KUKA KRL program: EPS_2_251520_SPSOVERFLOW_A_20260212031628.src

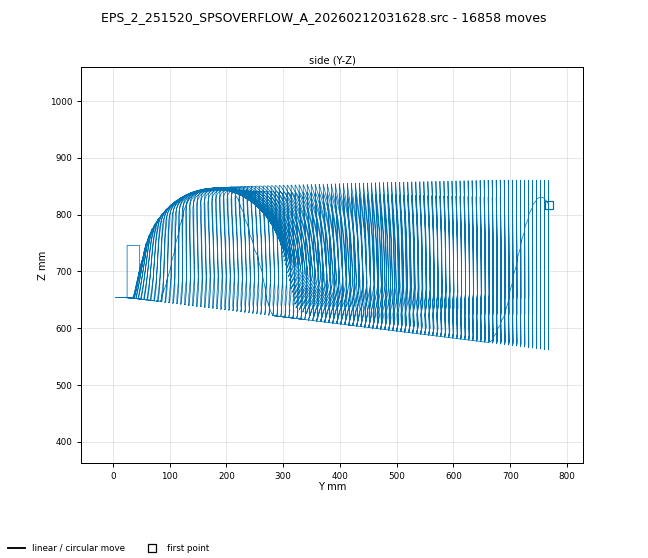
[picture p0: tool path of EPS_2_251520_SPSOVERFLOW_A_20260212031628.src, 16858 of 16860 moves have a stored position in this frame; points joined in program order, loops and branches not executed]
&ACCESS RVP
&REL 4
&COMMENT QRS 19112012
&PARAM EDITMASK = *
DEF PART()
EXT BAS (BAS_COMMAND :IN,REAL :IN )
INT I
BAS (#INITMOV,0 )

;KUKA QRS Post kuka4.cps  Date:22-06-2017 !

File_ID=3026

QRS_PRE_INIT()

;Init var - Until changes are made in qrs_pre_init
Outlet_Square_prg=0
Inlet_1_Square_prg=0
Inlet_2_Square_prg=0
Inlet_3_Square_prg=0
Inlet_4_Square_prg=0
Inlet_5_Square_prg=0

Outlet_1={X 0.000, Y 668.450, Z 760.500, B 0.000, E1 0.000 }
Inlet_1={X 0.000, Y 670.580, Z 730.500, B 0.000, E1 100.000 }
Outlet_1_type=201
Inlet_1_type=201
;QRS#1=Sidecore dimensions
;QRS#2=200-8" PVC SDR 35
;QRS#3=200-8" PVC SDR 35
;QRS#4=
;QRS#5=
;QRS#6=
;QRS#7=
;QRS#8=
;QRS#9=12-08 PSX
;QRS#10=12-08 PSX
;QRS#11=
;QRS#12=
;QRS#13=
;QRS#14=
;QRS#15=
;QRS#16=1524x152x1219 4'
;QRS#17=EPS Height
;QRS#18=861
;QRS#19=*
;QRS#20= UPDATED VERSION 22-06-2017
;QRS#21=*
Outlet_Square=0100
Inlet_1_Square=0100
Inlet_2_Square=0
Inlet_3_Square=0
Inlet_4_Square=0
Inlet_5_Square=0
Mill_Square=1
Outlet_Square_Prg=204
Inlet_1_Square_prg=204

QRS_INIT()

$ADVANCE=5

; T1
PTP {E1 174.142,E2 174.142}
PTP {X 0,Y 767.495,A -85,B 0,C 180,E1 174.142,E2 174.142,E3 0,E4 0,E5 0,E6 0}
QRS_SPEED_INIT()
LIN {X 0,Y 767.495,Z 817.254,A -85,B 0,C 180,E1 174.142,E2 174.142,E3 0,E4 0,E5 0,E6 0} C_VEL
LIN {X 0,Y 767.491,Z 822.732,A -85,B 0,C 180,E1 173.186,E2 173.186} C_VEL
LIN {X 0,Y 767.495,Z 825.01,A -85,B 0,C 180,E1 172.66,E2 172.66} C_VEL
LIN {X 0,Y 767.487,Z 828.448,A -85,B 0,C 180,E1 171.604,E2 171.604} C_VEL
LIN {X 0,Y 767.494,Z 830.063,A -85,B 0,C 180,E1 170.545,E2 170.545} C_VEL
LIN {X 0,Y 767.499,Z 830.375,A -85,B 0,C 180,E1 170.015,E2 170.015} C_VEL
LIN {X 0,Y 767.487,Z 829.609,A -85,B 0,C 180,E1 168.951,E2 168.951} C_VEL
LIN {X 0,Y 767.493,Z 828.662,A -85,B 0,C 180,E1 168.418,E2 168.418} C_VEL
LIN {X 0,Y 767.489,Z 825.435,A -85,B 0,C 180,E1 167.348,E2 167.348} C_VEL
LIN {X 0,Y 767.493,Z 821.811,A -85,B 0,C 180,E1 166.543,E2 166.543} C_VEL
LIN {X 0,Y 767.492,Z 817.014,A -85,B 0,C 180,E1 165.735,E2 165.735} C_VEL
LIN {X 0,Y 767.496,Z 810.871,A -85,B 0,C 180,E1 164.924,E2 164.924} C_VEL
LIN {X 0,Y 767.492,Z 804.595,A -85,B 0,C 180,E1 164.246,E2 164.246} C_VEL
LIN {X 0,Y 767.496,Z 796.955,A -85,B 0,C 180,E1 163.566,E2 163.566} C_VEL
LIN {X 0,Y 767.5,Z 788.629,A -85,B 0,C 180,E1 162.952,E2 162.952} C_VEL
LIN {X 0,Y 767.499,Z 780.947,A -85,B 0,C 180,E1 162.472,E2 162.472} C_VEL
LIN {X 0,Y 767.499,Z 771.732,A -85,B 0,C 180,E1 161.992,E2 161.992} C_VEL
LIN {X 0,Y 767.49,Z 762.141,A -85,B 0,C 180,E1 161.581,E2 161.581} C_VEL
LIN {X 0,Y 767.479,Z 750.832,A -85,B 0,C 180,E1 161.199,E2 161.199} C_VEL
LIN {X 0,Y 767.462,Z 740.016,A -85,B 0,C 180,E1 160.922,E2 160.922} C_VEL
LIN {X 0,Y 767.482,Z 729.744,A -85,B 0,C 180,E1 160.733,E2 160.733} C_VEL
LIN {X 0,Y 767.493,Z 712.465,A -85,B 0,C 180,E1 160.542,E2 160.542} C_VEL
LIN {X 0,Y 767.476,Z 620.271,A -85,B 0,C 180,E1 159.673,E2 159.673} C_VEL
LIN {X 0,Y 767.464,Z 604.056,A -85,B 0,C 180,E1 157.461,E2 157.461} C_VEL
LIN {X 0,Y 767.465,Z 586.448,A -85,B 0,C 180,E1 155.038,E2 155.038} C_VEL
LIN {X 0,Y 767.495,Z 568.677,A -85,B 0,C 180,E1 152.568,E2 152.568} C_VEL
LIN {X 0,Y 767.455,Z 561.691,A -85,B 0,C 180,E1 151.577,E2 151.577} C_VEL
LIN {X 0,Y 767.446,Z 561.687,A -85,B 0,C 180,E1 149.263,E2 149.263} C_VEL
LIN {X 0,Y 767.456,Z 561.684,A -85,B 0,C 180,E1 147.105,E2 147.105} C_VEL
LIN {X 0,Y 767.473,Z 561.68,A -85,B 0,C 180,E1 144.902,E2 144.902} C_VEL
LIN {X 0,Y 767.486,Z 561.692,A -85,B 0,C 180,E1 142.304,E2 142.304} C_VEL
LIN {X 0,Y 767.49,Z 561.702,A -85,B 0,C 180,E1 140.052,E2 140.052} C_VEL
LIN {X 0,Y 767.456,Z 561.69,A -85,B 0,C 180,E1 137.516,E2 137.516} C_VEL
LIN {X 0,Y 767.455,Z 561.686,A -85,B 0,C 180,E1 135.351,E2 135.351} C_VEL
LIN {X 0,Y 767.464,Z 561.682,A -85,B 0,C 180,E1 133.103,E2 133.103} C_VEL
LIN {X 0,Y 767.494,Z 561.677,A -85,B 0,C 180,E1 130.757,E2 130.757} C_VEL
LIN {X 0,Y 767.483,Z 561.693,A -85,B 0,C 180,E1 128.291,E2 128.291} C_VEL
LIN {X 0,Y 767.463,Z 561.693,A -85,B 0,C 180,E1 125.681,E2 125.681} C_VEL
LIN {X 0,Y 767.463,Z 561.683,A -85,B 0,C 180,E1 123.203,E2 123.203} C_VEL
LIN {X 0,Y 767.492,Z 561.678,A -85,B 0,C 180,E1 120.736,E2 120.736} C_VEL
LIN {X 0,Y 767.481,Z 561.692,A -85,B 0,C 180,E1 118.332,E2 118.332} C_VEL
LIN {X 0,Y 767.485,Z 561.7,A -85,B 0,C 180,E1 115.981,E2 115.981} C_VEL
LIN {X 0,Y 767.468,Z 561.691,A -85,B 0,C 180,E1 113.677,E2 113.677} C_VEL
LIN {X 0,Y 767.464,Z 561.685,A -85,B 0,C 180,E1 111.412,E2 111.412} C_VEL
LIN {X 0,Y 767.473,Z 561.68,A -85,B 0,C 180,E1 109.181,E2 109.181} C_VEL
LIN {X 0,Y 767.485,Z 561.677,A -85,B 0,C 180,E1 106.981,E2 106.981} C_VEL
LIN {X 0,Y 767.481,Z 561.682,A -85,B 0,C 180,E1 104.669,E2 104.669} C_VEL
LIN {X 0,Y 767.494,Z 561.698,A -85,B 0,C 180,E1 102.117,E2 102.117} C_VEL
LIN {X 0,Y 767.475,Z 561.691,A -85,B 0,C 180,E1 99.713,E2 99.713} C_VEL
LIN {X 0,Y 767.471,Z 561.682,A -85,B 0,C 180,E1 97.341,E2 97.341} C_VEL
LIN {X 0,Y 767.475,Z 561.68,A -85,B 0,C 180,E1 95.237,E2 95.237} C_VEL
LIN {X 0,Y 767.485,Z 561.677,A -85,B 0,C 180,E1 93.139,E2 93.139} C_VEL
LIN {X 0,Y 767.488,Z 561.676,A -85,B 0,C 180,E1 91.046,E2 91.046} C_VEL
LIN {X 0,Y 767.471,Z 561.69,A -85,B 0,C 180,E1 88.431,E2 88.431} C_VEL
LIN {X 0,Y 767.482,Z 561.693,A -85,B 0,C 180,E1 85.813,E2 85.813} C_VEL
LIN {X 0,Y 767.486,Z 561.677,A -85,B 0,C 180,E1 83.186,E2 83.186} C_VEL
LIN {X 0,Y 767.488,Z 561.676,A -85,B 0,C 180,E1 81.075,E2 81.075} C_VEL
LIN {X 0,Y 767.486,Z 561.677,A -85,B 0,C 180,E1 78.951,E2 78.951} C_VEL
LIN {X 0,Y 767.475,Z 561.681,A -85,B 0,C 180,E1 76.811,E2 76.811} C_VEL
LIN {X 0,Y 767.467,Z 561.685,A -85,B 0,C 180,E1 74.652,E2 74.652} C_VEL
LIN {X 0,Y 767.466,Z 561.69,A -85,B 0,C 180,E1 72.471,E2 72.471} C_VEL
LIN {X 0,Y 767.484,Z 561.704,A -85,B 0,C 180,E1 70.055,E2 70.055} C_VEL
LIN {X 0,Y 767.479,Z 561.683,A -85,B 0,C 180,E1 67.461,E2 67.461} C_VEL
LIN {X 0,Y 767.495,Z 561.675,A -85,B 0,C 180,E1 65.177,E2 65.177} C_VEL
LIN {X 0,Y 767.472,Z 561.681,A -85,B 0,C 180,E1 62.849,E2 62.849} C_VEL
LIN {X 0,Y 767.463,Z 561.691,A -85,B 0,C 180,E1 60.472,E2 60.472} C_VEL
LIN {X 0,Y 767.5,Z 561.699,A -85,B 0,C 180,E1 58.04,E2 58.04} C_VEL
LIN {X 0,Y 767.481,Z 561.684,A -85,B 0,C 180,E1 55.539,E2 55.539} C_VEL
LIN {X 0,Y 767.473,Z 561.68,A -85,B 0,C 180,E1 52.961,E2 52.961} C_VEL
LIN {X 0,Y 767.465,Z 561.682,A -85,B 0,C 180,E1 50.874,E2 50.874} C_VEL
LIN {X 0,Y 767.464,Z 561.692,A -85,B 0,C 180,E1 48.451,E2 48.451} C_VEL
LIN {X 0,Y 767.496,Z 561.7,A -85,B 0,C 180,E1 46.084,E2 46.084} C_VEL
LIN {X 0,Y 767.489,Z 561.693,A -85,B 0,C 180,E1 43.864,E2 43.864} C_VEL
LIN {X 0,Y 767.485,Z 561.683,A -85,B 0,C 180,E1 41.551,E2 41.551} C_VEL
LIN {X 0,Y 767.469,Z 561.681,A -85,B 0,C 180,E1 39.031,E2 39.031} C_VEL
LIN {X 0,Y 767.47,Z 561.68,A -85,B 0,C 180,E1 37.039,E2 37.039} C_VEL
LIN {X 0,Y 767.454,Z 561.686,A -85,B 0,C 180,E1 34.773,E2 34.773} C_VEL
LIN {X 0,Y 767.451,Z 561.691,A -85,B 0,C 180,E1 32.58,E2 32.58} C_VEL
LIN {X 0,Y 767.446,Z 561.689,A -85,B 0,C 180,E1 30.737,E2 30.737} C_VEL
LIN {X 0,Y 767.451,Z 561.686,A -85,B 0,C 180,E1 28.815,E2 28.815} C_VEL
LIN {X 0,Y 767.45,Z 561.692,A -85,B 0,C 180,E1 26.564,E2 26.564} C_VEL
LIN {X 0,Y 767.474,Z 561.697,A -85,B 0,C 180,E1 24.248,E2 24.248} C_VEL
LIN {X 0,Y 767.489,Z 561.698,A -85,B 0,C 180,E1 21.974,E2 21.974} C_VEL
LIN {X 0,Y 767.489,Z 561.688,A -85,B 0,C 180,E1 19.735,E2 19.735} C_VEL
LIN {X 0,Y 767.491,Z 561.682,A -85,B 0,C 180,E1 17.528,E2 17.528} C_VEL
LIN {X 0,Y 767.485,Z 561.679,A -85,B 0,C 180,E1 15.347,E2 15.347} C_VEL
LIN {X 0,Y 767.468,Z 561.681,A -85,B 0,C 180,E1 13.189,E2 13.189} C_VEL
LIN {X 0,Y 767.453,Z 561.684,A -85,B 0,C 180,E1 11.05,E2 11.05} C_VEL
LIN {X 0,Y 767.446,Z 561.686,A -85,B 0,C 180,E1 8.926,E2 8.926} C_VEL
LIN {X 0,Y 767.44,Z 561.689,A -85,B 0,C 180,E1 6.814,E2 6.814} C_VEL
LIN {X 0,Y 767.437,Z 561.691,A -85,B 0,C 180,E1 4.712,E2 4.712} C_VEL
LIN {X 0,Y 767.438,Z 561.693,A -85,B 0,C 180,E1 2.615,E2 2.615} C_VEL
LIN {X 0,Y 767.445,Z 561.694,A -85,B 0,C 180,E1 0.523,E2 0.523} C_VEL
LIN {X 0,Y 767.448,Z 561.696,A -85,B 0,C 180,E1 -1.569,E2 -1.569} C_VEL
LIN {X 0,Y 767.455,Z 561.698,A -85,B 0,C 180,E1 -3.663,E2 -3.663} C_VEL
LIN {X 0,Y 767.493,Z 561.687,A -85,B 0,C 180,E1 -6.288,E2 -6.288} C_VEL
LIN {X 0,Y 767.495,Z 561.682,A -85,B 0,C 180,E1 -8.397,E2 -8.397} C_VEL
LIN {X 0,Y 767.481,Z 561.683,A -85,B 0,C 180,E1 -10.517,E2 -10.517} C_VEL
LIN {X 0,Y 767.466,Z 561.684,A -85,B 0,C 180,E1 -12.653,E2 -12.653} C_VEL
LIN {X 0,Y 767.447,Z 561.686,A -85,B 0,C 180,E1 -14.807,E2 -14.807} C_VEL
LIN {X 0,Y 767.432,Z 561.689,A -85,B 0,C 180,E1 -16.982,E2 -16.982} C_VEL
LIN {X 0,Y 767.463,Z 561.684,A -85,B 0,C 180,E1 -18.629,E2 -18.629} C_VEL
LIN {X 0,Y 767.434,Z 561.689,A -85,B 0,C 180,E1 -20.852,E2 -20.852} C_VEL
LIN {X 0,Y 767.441,Z 561.688,A -85,B 0,C 180,E1 -22.805,E2 -22.805} C_VEL
LIN {X 0,Y 767.437,Z 561.688,A -85,B 0,C 180,E1 -24.825,E2 -24.825} C_VEL
LIN {X 0,Y 767.465,Z 561.685,A -85,B 0,C 180,E1 -26.566,E2 -26.566} C_VEL
LIN {X 0,Y 767.425,Z 561.691,A -85,B 0,C 180,E1 -28.93,E2 -28.93} C_VEL
LIN {X 0,Y 767.427,Z 561.69,A -85,B 0,C 180,E1 -30.912,E2 -30.912} C_VEL
LIN {X 0,Y 767.428,Z 561.69,A -85,B 0,C 180,E1 -32.892,E2 -32.892} C_VEL
LIN {X 0,Y 767.419,Z 561.693,A -85,B 0,C 180,E1 -35.101,E2 -35.101} C_VEL
LIN {X 0,Y 767.417,Z 561.693,A -85,B 0,C 180,E1 -37.042,E2 -37.042} C_VEL
LIN {X 0,Y 767.416,Z 561.694,A -85,B 0,C 180,E1 -39.12,E2 -39.12} C_VEL
LIN {X 0,Y 767.414,Z 561.694,A -85,B 0,C 180,E1 -41.084,E2 -41.084} C_VEL
LIN {X 0,Y 767.412,Z 561.695,A -85,B 0,C 180,E1 -43.2,E2 -43.2} C_VEL
LIN {X 0,Y 767.439,Z 561.69,A -85,B 0,C 180,E1 -44.651,E2 -44.651} C_VEL
LIN {X 0,Y 767.424,Z 561.691,A -85,B 0,C 180,E1 -46.801,E2 -46.801} C_VEL
LIN {X 0,Y 767.414,Z 561.693,A -85,B 0,C 180,E1 -48.916,E2 -48.916} C_VEL
LIN {X 0,Y 767.414,Z 561.693,A -85,B 0,C 180,E1 -50.88,E2 -50.88} C_VEL
LIN {X 0,Y 767.412,Z 561.694,A -85,B 0,C 180,E1 -52.958,E2 -52.958} C_VEL
LIN {X 0,Y 767.412,Z 561.694,A -85,B 0,C 180,E1 -54.899,E2 -54.899} C_VEL
LIN {X 0,Y 767.415,Z 561.693,A -85,B 0,C 180,E1 -56.795,E2 -56.795} C_VEL
LIN {X 0,Y 767.426,Z 561.693,A -85,B 0,C 180,E1 -58.651,E2 -58.651} C_VEL
LIN {X 0,Y 767.446,Z 561.692,A -85,B 0,C 180,E1 -60.472,E2 -60.472} C_VEL
LIN {X 0,Y 767.407,Z 561.695,A -85,B 0,C 180,E1 -62.847,E2 -62.847} C_VEL
LIN {X 0,Y 767.422,Z 561.694,A -85,B 0,C 180,E1 -64.635,E2 -64.635} C_VEL
LIN {X 0,Y 767.463,Z 561.692,A -85,B 0,C 180,E1 -66.323,E2 -66.323} C_VEL
LIN {X 0,Y 767.424,Z 561.694,A -85,B 0,C 180,E1 -68.587,E2 -68.587} C_VEL
LIN {X 0,Y 767.421,Z 561.842,A -85,B 0,C 180,E1 -69.427,E2 -69.427} C_VEL
LIN {X 0,Y 767.495,Z 582.633,A -85,B 0,C 180,E1 -71.923,E2 -71.923} C_VEL
LIN {X 0,Y 767.459,Z 604.567,A -85,B 0,C 180,E1 -74.517,E2 -74.517} C_VEL
LIN {X 0,Y 767.47,Z 624.17,A -85,B 0,C 180,E1 -76.811,E2 -76.811} C_VEL
LIN {X 0,Y 767.443,Z 643.774,A -85,B 0,C 180,E1 -79.083,E2 -79.083} C_VEL
LIN {X 0,Y 767.461,Z 649.237,A -85,B 0,C 180,E1 -79.715,E2 -79.715} C_VEL
LIN {X 0,Y 767.441,Z 755.809,A -85,B 0,C 180,E1 -80.727,E2 -80.727} C_VEL
LIN {X 0,Y 767.444,Z 765.448,A -85,B 0,C 180,E1 -80.876,E2 -80.876} C_VEL
LIN {X 0,Y 767.459,Z 775.895,A -85,B 0,C 180,E1 -81.107,E2 -81.107} C_VEL
LIN {X 0,Y 767.494,Z 785.992,A -85,B 0,C 180,E1 -81.405,E2 -81.405} C_VEL
LIN {X 0,Y 767.491,Z 796.476,A -85,B 0,C 180,E1 -81.802,E2 -81.802} C_VEL
LIN {X 0,Y 767.491,Z 806.3,A -85,B 0,C 180,E1 -82.264,E2 -82.264} C_VEL
LIN {X 0,Y 767.498,Z 815.493,A -85,B 0,C 180,E1 -82.791,E2 -82.791} C_VEL
LIN {X 0,Y 767.498,Z 823.204,A -85,B 0,C 180,E1 -83.318,E2 -83.318} C_VEL
LIN {X 0,Y 767.496,Z 830.667,A -85,B 0,C 180,E1 -83.925,E2 -83.925} C_VEL
LIN {X 0,Y 767.494,Z 837.879,A -85,B 0,C 180,E1 -84.632,E2 -84.632} C_VEL
LIN {X 0,Y 767.491,Z 843.46,A -85,B 0,C 180,E1 -85.289,E2 -85.289} C_VEL
LIN {X 0,Y 767.496,Z 848.873,A -85,B 0,C 180,E1 -86.075,E2 -86.075} C_VEL
LIN {X 0,Y 767.491,Z 853.131,A -85,B 0,C 180,E1 -86.861,E2 -86.861} C_VEL
LIN {X 0,Y 767.491,Z 855.399,A -85,B 0,C 180,E1 -87.385,E2 -87.385} C_VEL
LIN {X 0,Y 767.488,Z 858.607,A -85,B 0,C 180,E1 -88.431,E2 -88.431} C_VEL
LIN {X 0,Y 767.491,Z 860.103,A -85,B 0,C 180,E1 -89.477,E2 -89.477} C_VEL
LIN {X 0,Y 767.491,Z 860.39,A -85,B 0,C 180,E1 -90,E2 -90} C_VEL
LIN {X 0,Y 767.487,Z 859.535,A -85,B 0,C 180,E1 -91.046,E2 -91.046} C_VEL
LIN {X 0,Y 767.488,Z 858.607,A -85,B 0,C 180,E1 -91.569,E2 -91.569} C_VEL
LIN {X 0,Y 767.491,Z 855.398,A -85,B 0,C 180,E1 -92.616,E2 -92.616} C_VEL
LIN {X 0,Y 767.492,Z 851.876,A -85,B 0,C 180,E1 -93.401,E2 -93.401} C_VEL
LIN {X 0,Y 767.493,Z 847.253,A -85,B 0,C 180,E1 -94.187,E2 -94.187} C_VEL
LIN {X 0,Y 767.496,Z 841.377,A -85,B 0,C 180,E1 -94.974,E2 -94.974} C_VEL
LIN {X 0,Y 767.493,Z 834.027,A -85,B 0,C 180,E1 -95.762,E2 -95.762} C_VEL
LIN {X 0,Y 767.497,Z 826.571,A -85,B 0,C 180,E1 -96.419,E2 -96.419} C_VEL
LIN {X 0,Y 767.497,Z 819.513,A -85,B 0,C 180,E1 -96.946,E2 -96.946} C_VEL
LIN {X 0,Y 767.495,Z 811.13,A -85,B 0,C 180,E1 -97.473,E2 -97.473} C_VEL
LIN {X 0,Y 767.493,Z 802.375,A -85,B 0,C 180,E1 -97.934,E2 -97.934} C_VEL
LIN {X 0,Y 767.491,Z 791.513,A -85,B 0,C 180,E1 -98.397,E2 -98.397} C_VEL
LIN {X 0,Y 767.477,Z 781.86,A -85,B 0,C 180,E1 -98.727,E2 -98.727} C_VEL
LIN {X 0,Y 767.449,Z 770.388,A -85,B 0,C 180,E1 -99.025,E2 -99.025} C_VEL
LIN {X 0,Y 767.441,Z 759.668,A -85,B 0,C 180,E1 -99.224,E2 -99.224} C_VEL
LIN {X 0,Y 767.443,Z 741.469,A -85,B 0,C 180,E1 -99.423,E2 -99.423} C_VEL
LIN {X 0,Y 767.461,Z 649.235,A -85,B 0,C 180,E1 -100.285,E2 -100.285} C_VEL
LIN {X 0,Y 767.483,Z 628.781,A -85,B 0,C 180,E1 -102.653,E2 -102.653} C_VEL
LIN {X 0,Y 767.439,Z 609.18,A -85,B 0,C 180,E1 -104.942,E2 -104.942} C_VEL
LIN {X 0,Y 767.495,Z 589.556,A -85,B 0,C 180,E1 -107.254,E2 -107.254} C_VEL
LIN {X 0,Y 767.475,Z 568.772,A -85,B 0,C 180,E1 -109.736,E2 -109.736} C_VEL
LIN {X 0,Y 767.416,Z 561.699,A -85,B 0,C 180,E1 -110.608,E2 -110.608} C_VEL
LIN {X 0,Y 767.418,Z 561.699,A -85,B 0,C 180,E1 -112.541,E2 -112.541} C_VEL
LIN {X 0,Y 767.454,Z 561.698,A -85,B 0,C 180,E1 -114.25,E2 -114.25} C_VEL
LIN {X 0,Y 767.417,Z 561.696,A -85,B 0,C 180,E1 -116.567,E2 -116.567} C_VEL
LIN {X 0,Y 767.445,Z 561.693,A -85,B 0,C 180,E1 -118.334,E2 -118.334} C_VEL
LIN {X 0,Y 767.473,Z 561.691,A -85,B 0,C 180,E1 -120.13,E2 -120.13} C_VEL
LIN {X 0,Y 767.428,Z 561.692,A -85,B 0,C 180,E1 -122.582,E2 -122.582} C_VEL
LIN {X 0,Y 767.44,Z 561.69,A -85,B 0,C 180,E1 -124.463,E2 -124.463} C_VEL
LIN {X 0,Y 767.437,Z 561.69,A -85,B 0,C 180,E1 -126.565,E2 -126.565} C_VEL
LIN {X 0,Y 767.454,Z 561.686,A -85,B 0,C 180,E1 -128.362,E2 -128.362} C_VEL
LIN {X 0,Y 767.454,Z 561.686,A -85,B 0,C 180,E1 -130.392,E2 -130.392} C_VEL
LIN {X 0,Y 767.452,Z 561.687,A -85,B 0,C 180,E1 -132.485,E2 -132.485} C_VEL
LIN {X 0,Y 767.451,Z 561.689,A -85,B 0,C 180,E1 -134.65,E2 -134.65} C_VEL
LIN {X 0,Y 767.466,Z 561.694,A -85,B 0,C 180,E1 -136.898,E2 -136.898} C_VEL
LIN {X 0,Y 767.493,Z 561.698,A -85,B 0,C 180,E1 -139.244,E2 -139.244} C_VEL
LIN {X 0,Y 767.487,Z 561.682,A -85,B 0,C 180,E1 -141.71,E2 -141.71} C_VEL
LIN {X 0,Y 767.474,Z 561.683,A -85,B 0,C 180,E1 -144.26,E2 -144.26} C_VEL
LIN {X 0,Y 767.488,Z 561.697,A -85,B 0,C 180,E1 -146.798,E2 -146.798} C_VEL
LIN {X 0,Y 767.467,Z 561.691,A -85,B 0,C 180,E1 -149.263,E2 -149.263} C_VEL
LIN {X 0,Y 767.498,Z 561.676,A -85,B 0,C 180,E1 -151.669,E2 -151.669} C_VEL
LIN {X 0,Y 767.492,Z 561.68,A -85,B 0,C 180,E1 -154.019,E2 -154.019} C_VEL
LIN {X 0,Y 767.487,Z 561.69,A -85,B 0,C 180,E1 -156.324,E2 -156.324} C_VEL
LIN {X 0,Y 767.493,Z 561.7,A -85,B 0,C 180,E1 -158.589,E2 -158.589} C_VEL
LIN {X 0,Y 767.459,Z 561.696,A -85,B 0,C 180,E1 -160.818,E2 -160.818} C_VEL
LIN {X 0,Y 767.439,Z 561.693,A -85,B 0,C 180,E1 -163.018,E2 -163.018} C_VEL
LIN {X 0,Y 767.447,Z 561.688,A -85,B 0,C 180,E1 -165.193,E2 -165.193} C_VEL
LIN {X 0,Y 767.493,Z 561.679,A -85,B 0,C 180,E1 -167.562,E2 -167.562} C_VEL
LIN {X 0,Y 767.477,Z 561.701,A -85,B 0,C 180,E1 -170.29,E2 -170.29} C_VEL
LIN {X 0,Y 767.493,Z 561.864,A -85,B 0,C 180,E1 -171.702,E2 -171.702} C_VEL
LIN {X 0,Y 767.494,Z 580.016,A -85,B 0,C 180,E1 -174.238,E2 -174.238} C_VEL
LIN {X 0,Y 767.486,Z 597.113,A -85,B 0,C 180,E1 -176.599,E2 -176.599} C_VEL
LIN {X 0,Y 767.477,Z 614.326,A -85,B 0,C 180,E1 -178.954,E2 -178.954} C_VEL
LIN {X 0,Y 767.493,Z 620.326,A -85,B 0,C 180,E1 -179.771,E2 -179.771} C_VEL
LIN {X 0,Y 767.462,Z 725.497,A -85,B 0,C 180,E1 -180.768,E2 -180.768} C_VEL
LIN {X 0,Y 767.461,Z 735.156,A -85,B 0,C 180,E1 -180.915,E2 -180.915} C_VEL
LIN {X 0,Y 767.468,Z 745.579,A -85,B 0,C 180,E1 -181.144,E2 -181.144} C_VEL
LIN {X 0,Y 767.487,Z 755.65,A -85,B 0,C 180,E1 -181.438,E2 -181.438} C_VEL
LIN {X 0,Y 767.49,Z 766.109,A -85,B 0,C 180,E1 -181.83,E2 -181.83} C_VEL
LIN {X 0,Y 767.492,Z 775.922,A -85,B 0,C 180,E1 -182.288,E2 -182.288} C_VEL
LIN {X 0,Y 767.499,Z 784.117,A -85,B 0,C 180,E1 -182.746,E2 -182.746} C_VEL
LIN {X 0,Y 767.497,Z 793.687,A -85,B 0,C 180,E1 -183.401,E2 -183.401} C_VEL
LIN {X 0,Y 767.496,Z 800.181,A -85,B 0,C 180,E1 -183.925,E2 -183.925} C_VEL
LIN {X 0,Y 767.492,Z 807.015,A -85,B 0,C 180,E1 -184.58,E2 -184.58} C_VEL
LIN {X 0,Y 767.49,Z 812.754,A -85,B 0,C 180,E1 -185.236,E2 -185.236} C_VEL
LIN {X 0,Y 767.495,Z 817.254,A -85,B 0,C 180,E1 -185.858,E2 -185.858} C_VEL
LIN {X 0,Y 766.834,Z 819.82,A -85,B 0,C 180,E1 -186.257,E2 -186.257} C_VEL
LIN {X 0,Y 764.632,Z 823.081,A -85,B 0,C 180,E1 -186.779,E2 -186.779} C_VEL
LIN {X 0,Y 761.57,Z 826.138,A -85,B 0,C 180,E1 -187.448,E2 -187.448} C_VEL
LIN {X 0,Y 760.517,Z 827.544,A -85,B 0,C 180,E1 -187.871,E2 -187.871} C_VEL
LIN {X 0,Y 760.425,Z 827.957,A -85,B 0,C 180,E1 -188.016,E2 -188.016} C_VEL
LIN {X 0,Y 760.415,Z 829.23,A -85,B 0,C 180,E1 -188.475,E2 -188.475} C_VEL
LIN {X 0,Y 760.44,Z 830.176,A -85,B 0,C 180,E1 -189.009,E2 -189.009} C_VEL
LIN {X 0,Y 760.425,Z 830.996,A -85,B 0,C 180,E1 -190.079,E2 -190.079} C_VEL
LIN {X 0,Y 760.428,Z 830.049,A -85,B 0,C 180,E1 -191.153,E2 -191.153} C_VEL
LIN {X 0,Y 760.442,Z 829.081,A -85,B 0,C 180,E1 -191.691,E2 -191.691} C_VEL
LIN {X 0,Y 760.433,Z 826.759,A -85,B 0,C 180,E1 -192.477,E2 -192.477} C_VEL
LIN {X 0,Y 760.44,Z 823.257,A -85,B 0,C 180,E1 -193.313,E2 -193.313} C_VEL
LIN {X 0,Y 760.448,Z 818.707,A -85,B 0,C 180,E1 -194.128,E2 -194.128} C_VEL
LIN {X 0,Y 760.442,Z 811.706,A -85,B 0,C 180,E1 -195.082,E2 -195.082} C_VEL
LIN {X 0,Y 760.455,Z 805.469,A -85,B 0,C 180,E1 -195.766,E2 -195.766} C_VEL
LIN {X 0,Y 760.468,Z 797.88,A -85,B 0,C 180,E1 -196.453,E2 -196.453} C_VEL
LIN {X 0,Y 760.475,Z 789.604,A -85,B 0,C 180,E1 -197.074,E2 -197.074} C_VEL
LIN {X 0,Y 760.463,Z 780.774,A -85,B 0,C 180,E1 -197.626,E2 -197.626} C_VEL
LIN {X 0,Y 760.478,Z 771.423,A -85,B 0,C 180,E1 -198.111,E2 -198.111} C_VEL
LIN {X 0,Y 760.484,Z 762.477,A -85,B 0,C 180,E1 -198.496,E2 -198.496} C_VEL
LIN {X 0,Y 760.471,Z 751.37,A -85,B 0,C 180,E1 -198.876,E2 -198.876} C_VEL
LIN {X 0,Y 760.462,Z 739.812,A -85,B 0,C 180,E1 -199.173,E2 -199.173} C_VEL
LIN {X 0,Y 760.498,Z 729.365,A -85,B 0,C 180,E1 -199.364,E2 -199.364} C_VEL
LIN {X 0,Y 760.522,Z 711.856,A -85,B 0,C 180,E1 -199.556,E2 -199.556} C_VEL
LIN {X 0,Y 760.453,Z 620.552,A -85,B 0,C 180,E1 -200.422,E2 -200.422} C_VEL
LIN {X 0,Y 760.436,Z 603.516,A -85,B 0,C 180,E1 -202.759,E2 -202.759} C_VEL
LIN {X 0,Y 760.451,Z 587.883,A -85,B 0,C 180,E1 -204.923,E2 -204.923} C_VEL
LIN {X 0,Y 760.473,Z 571.077,A -85,B 0,C 180,E1 -207.273,E2 -207.273} C_VEL
LIN {X 0,Y 760.439,Z 562.69,A -85,B 0,C 180,E1 -208.468,E2 -208.468} C_VEL
LIN {X 0,Y 760.423,Z 562.692,A -85,B 0,C 180,E1 -210.438,E2 -210.438} C_VEL
LIN {X 0,Y 760.434,Z 562.693,A -85,B 0,C 180,E1 -212.292,E2 -212.292} C_VEL
LIN {X 0,Y 760.444,Z 562.694,A -85,B 0,C 180,E1 -214.185,E2 -214.185} C_VEL
LIN {X 0,Y 760.437,Z 562.686,A -85,B 0,C 180,E1 -216.778,E2 -216.778} C_VEL
LIN {X 0,Y 760.464,Z 562.684,A -85,B 0,C 180,E1 -219.312,E2 -219.312} C_VEL
LIN {X 0,Y 760.46,Z 562.692,A -85,B 0,C 180,E1 -221.748,E2 -221.748} C_VEL
LIN {X 0,Y 760.444,Z 562.696,A -85,B 0,C 180,E1 -224.072,E2 -224.072} C_VEL
LIN {X 0,Y 760.453,Z 562.69,A -85,B 0,C 180,E1 -226.305,E2 -226.305} C_VEL
LIN {X 0,Y 760.45,Z 562.688,A -85,B 0,C 180,E1 -228.456,E2 -228.456} C_VEL
LIN {X 0,Y 760.453,Z 562.685,A -85,B 0,C 180,E1 -230.688,E2 -230.688} C_VEL
LIN {X 0,Y 760.459,Z 562.685,A -85,B 0,C 180,E1 -233.258,E2 -233.258} C_VEL
LIN {X 0,Y 760.453,Z 562.697,A -85,B 0,C 180,E1 -235.993,E2 -235.993} C_VEL
LIN {X 0,Y 760.458,Z 562.689,A -85,B 0,C 180,E1 -238.33,E2 -238.33} C_VEL
LIN {X 0,Y 760.442,Z 562.686,A -85,B 0,C 180,E1 -240.779,E2 -240.779} C_VEL
LIN {X 0,Y 760.468,Z 562.684,A -85,B 0,C 180,E1 -243.307,E2 -243.307} C_VEL
LIN {X 0,Y 760.46,Z 562.693,A -85,B 0,C 180,E1 -245.764,E2 -245.764} C_VEL
LIN {X 0,Y 760.475,Z 562.692,A -85,B 0,C 180,E1 -247.813,E2 -247.813} C_VEL
LIN {X 0,Y 760.478,Z 562.692,A -85,B 0,C 180,E1 -250.075,E2 -250.075} C_VEL
LIN {X 0,Y 760.449,Z 562.691,A -85,B 0,C 180,E1 -252.304,E2 -252.304} C_VEL
LIN {X 0,Y 760.451,Z 562.687,A -85,B 0,C 180,E1 -254.507,E2 -254.507} C_VEL
LIN {X 0,Y 760.44,Z 562.687,A -85,B 0,C 180,E1 -256.687,E2 -256.687} C_VEL
LIN {X 0,Y 760.45,Z 562.685,A -85,B 0,C 180,E1 -258.847,E2 -258.847} C_VEL
LIN {X 0,Y 760.47,Z 562.682,A -85,B 0,C 180,E1 -260.991,E2 -260.991} C_VEL
LIN {X 0,Y 760.45,Z 562.692,A -85,B 0,C 180,E1 -263.654,E2 -263.654} C_VEL
LIN {X 0,Y 760.456,Z 562.694,A -85,B 0,C 180,E1 -265.774,E2 -265.774} C_VEL
LIN {X 0,Y 760.479,Z 562.694,A -85,B 0,C 180,E1 -267.889,E2 -267.889} C_VEL
LIN {X 0,Y 760.471,Z 562.684,A -85,B 0,C 180,E1 -270.528,E2 -270.528} C_VEL
LIN {X 0,Y 760.456,Z 562.685,A -85,B 0,C 180,E1 -272.64,E2 -272.64} C_VEL
LIN {X 0,Y 760.474,Z 562.683,A -85,B 0,C 180,E1 -275.285,E2 -275.285} C_VEL
LIN {X 0,Y 760.441,Z 562.689,A -85,B 0,C 180,E1 -277.409,E2 -277.409} C_VEL
LIN {X 0,Y 760.454,Z 562.693,A -85,B 0,C 180,E1 -279.751,E2 -279.751} C_VEL
LIN {X 0,Y 760.476,Z 562.689,A -85,B 0,C 180,E1 -282.23,E2 -282.23} C_VEL
LIN {X 0,Y 760.459,Z 562.683,A -85,B 0,C 180,E1 -284.946,E2 -284.946} C_VEL
LIN {X 0,Y 760.454,Z 562.684,A -85,B 0,C 180,E1 -287.142,E2 -287.142} C_VEL
LIN {X 0,Y 760.448,Z 562.687,A -85,B 0,C 180,E1 -289.365,E2 -289.365} C_VEL
LIN {X 0,Y 760.456,Z 562.69,A -85,B 0,C 180,E1 -291.619,E2 -291.619} C_VEL
LIN {X 0,Y 760.445,Z 562.698,A -85,B 0,C 180,E1 -293.909,E2 -293.909} C_VEL
LIN {X 0,Y 760.461,Z 562.69,A -85,B 0,C 180,E1 -296.239,E2 -296.239} C_VEL
LIN {X 0,Y 760.452,Z 562.686,A -85,B 0,C 180,E1 -298.618,E2 -298.618} C_VEL
LIN {X 0,Y 760.454,Z 562.684,A -85,B 0,C 180,E1 -301.063,E2 -301.063} C_VEL
LIN {X 0,Y 760.461,Z 562.688,A -85,B 0,C 180,E1 -303.549,E2 -303.549} C_VEL
LIN {X 0,Y 760.448,Z 562.694,A -85,B 0,C 180,E1 -306.121,E2 -306.121} C_VEL
LIN {X 0,Y 760.456,Z 562.684,A -85,B 0,C 180,E1 -308.78,E2 -308.78} C_VEL
LIN {X 0,Y 760.466,Z 562.682,A -85,B 0,C 180,E1 -310.951,E2 -310.951} C_VEL
LIN {X 0,Y 760.445,Z 562.687,A -85,B 0,C 180,E1 -313.309,E2 -313.309} C_VEL
LIN {X 0,Y 760.426,Z 562.693,A -85,B 0,C 180,E1 -315.569,E2 -315.569} C_VEL
LIN {X 0,Y 760.435,Z 562.696,A -85,B 0,C 180,E1 -317.747,E2 -317.747} C_VEL
LIN {X 0,Y 760.468,Z 562.694,A -85,B 0,C 180,E1 -319.861,E2 -319.861} C_VEL
LIN {X 0,Y 760.463,Z 562.685,A -85,B 0,C 180,E1 -322.562,E2 -322.562} C_VEL
LIN {X 0,Y 760.432,Z 562.687,A -85,B 0,C 180,E1 -325.174,E2 -325.174} C_VEL
LIN {X 0,Y 760.436,Z 562.686,A -85,B 0,C 180,E1 -327.081,E2 -327.081} C_VEL
LIN {X 0,Y 760.449,Z 562.684,A -85,B 0,C 180,E1 -328.949,E2 -328.949} C_VEL
LIN {X 0,Y 760.422,Z 562.691,A -85,B 0,C 180,E1 -331.381,E2 -331.381} C_VEL
LIN {X 0,Y 760.449,Z 562.694,A -85,B 0,C 180,E1 -333.761,E2 -333.761} C_VEL
LIN {X 0,Y 760.454,Z 562.694,A -85,B 0,C 180,E1 -336.092,E2 -336.092} C_VEL
LIN {X 0,Y 760.473,Z 562.685,A -85,B 0,C 180,E1 -338.478,E2 -338.478} C_VEL
LIN {X 0,Y 760.452,Z 562.686,A -85,B 0,C 180,E1 -340.635,E2 -340.635} C_VEL
LIN {X 0,Y 760.443,Z 562.685,A -85,B 0,C 180,E1 -342.858,E2 -342.858} C_VEL
LIN {X 0,Y 760.43,Z 562.688,A -85,B 0,C 180,E1 -345.278,E2 -345.278} C_VEL
LIN {X 0,Y 760.468,Z 562.692,A -85,B 0,C 180,E1 -347.77,E2 -347.77} C_VEL
LIN {X 0,Y 760.474,Z 562.685,A -85,B 0,C 180,E1 -350.457,E2 -350.457} C_VEL
LIN {X 0,Y 760.452,Z 562.686,A -85,B 0,C 180,E1 -352.591,E2 -352.591} C_VEL
LIN {X 0,Y 760.444,Z 562.686,A -85,B 0,C 180,E1 -354.715,E2 -354.715} C_VEL
LIN {X 0,Y 760.424,Z 562.688,A -85,B 0,C 180,E1 -356.832,E2 -356.832} C_VEL
LIN {X 0,Y 760.437,Z 562.686,A -85,B 0,C 180,E1 -358.945,E2 -358.945} C_VEL
LIN {X 0,Y 760.43,Z 562.687,A -85,B 0,C 180,E1 -361.056,E2 -361.056} C_VEL
LIN {X 0,Y 760.406,Z 562.691,A -85,B 0,C 180,E1 -363.168,E2 -363.168} C_VEL
LIN {X 0,Y 760.413,Z 562.691,A -85,B 0,C 180,E1 -365.285,E2 -365.285} C_VEL
LIN {X 0,Y 760.409,Z 562.693,A -85,B 0,C 180,E1 -367.41,E2 -367.41} C_VEL
LIN {X 0,Y 760.44,Z 562.695,A -85,B 0,C 180,E1 -369.741,E2 -369.741} C_VEL
LIN {X 0,Y 760.486,Z 562.687,A -85,B 0,C 180,E1 -372.23,E2 -372.23} C_VEL
LIN {X 0,Y 760.434,Z 562.686,A -85,B 0,C 180,E1 -374.946,E2 -374.946} C_VEL
LIN {X 0,Y 760.417,Z 562.689,A -85,B 0,C 180,E1 -377.143,E2 -377.143} C_VEL
LIN {X 0,Y 760.425,Z 562.688,A -85,B 0,C 180,E1 -378.808,E2 -378.808} C_VEL
LIN {X 0,Y 760.454,Z 562.687,A -85,B 0,C 180,E1 -380.488,E2 -380.488} C_VEL
LIN {X 0,Y 760.404,Z 562.69,A -85,B 0,C 180,E1 -382.906,E2 -382.906} C_VEL
LIN {X 0,Y 760.396,Z 562.691,A -85,B 0,C 180,E1 -385.07,E2 -385.07} C_VEL
LIN {X 0,Y 760.409,Z 562.69,A -85,B 0,C 180,E1 -386.831,E2 -386.831} C_VEL
LIN {X 0,Y 760.404,Z 562.69,A -85,B 0,C 180,E1 -388.944,E2 -388.944} C_VEL
LIN {X 0,Y 760.393,Z 562.692,A -85,B 0,C 180,E1 -391.054,E2 -391.054} C_VEL
LIN {X 0,Y 760.41,Z 562.69,A -85,B 0,C 180,E1 -393.046,E2 -393.046} C_VEL
LIN {X 0,Y 760.397,Z 562.691,A -85,B 0,C 180,E1 -394.932,E2 -394.932} C_VEL
LIN {X 0,Y 760.427,Z 562.688,A -85,B 0,C 180,E1 -396.779,E2 -396.779} C_VEL
LIN {X 0,Y 760.423,Z 562.688,A -85,B 0,C 180,E1 -398.782,E2 -398.782} C_VEL
LIN {X 0,Y 760.412,Z 562.689,A -85,B 0,C 180,E1 -400.946,E2 -400.946} C_VEL
LIN {X 0,Y 760.408,Z 562.692,A -85,B 0,C 180,E1 -403.306,E2 -403.306} C_VEL
LIN {X 0,Y 760.442,Z 562.7,A -85,B 0,C 180,E1 -405.927,E2 -405.927} C_VEL
LIN {X 0,Y 760.452,Z 562.688,A -85,B 0,C 180,E1 -408.457,E2 -408.457} C_VEL
LIN {X 0,Y 760.414,Z 562.69,A -85,B 0,C 180,E1 -410.692,E2 -410.692} C_VEL
LIN {X 0,Y 760.414,Z 562.691,A -85,B 0,C 180,E1 -412.559,E2 -412.559} C_VEL
LIN {X 0,Y 760.417,Z 562.691,A -85,B 0,C 180,E1 -414.528,E2 -414.528} C_VEL
LIN {X 0,Y 760.422,Z 562.691,A -85,B 0,C 180,E1 -416.449,E2 -416.449} C_VEL
LIN {X 0,Y 760.449,Z 562.69,A -85,B 0,C 180,E1 -418.33,E2 -418.33} C_VEL
LIN {X 0,Y 760.401,Z 562.691,A -85,B 0,C 180,E1 -420.777,E2 -420.777} C_VEL
LIN {X 0,Y 760.426,Z 562.689,A -85,B 0,C 180,E1 -422.577,E2 -422.577} C_VEL
LIN {X 0,Y 760.43,Z 562.69,A -85,B 0,C 180,E1 -424.514,E2 -424.514} C_VEL
LIN {X 0,Y 760.403,Z 562.692,A -85,B 0,C 180,E1 -426.666,E2 -426.666} C_VEL
LIN {X 0,Y 760.373,Z 562.695,A -85,B 0,C 180,E1 -428.945,E2 -428.945} C_VEL
LIN {X 0,Y 760.398,Z 562.723,A -85,B 0,C 180,E1 -429.334,E2 -429.334} C_VEL
LIN {X 0,Y 760.497,Z 578.051,A -85,B 0,C 180,E1 -431.194,E2 -431.194} C_VEL
LIN {X 0,Y 760.474,Z 597.717,A -85,B 0,C 180,E1 -433.547,E2 -433.547} C_VEL
LIN {X 0,Y 760.478,Z 619.697,A -85,B 0,C 180,E1 -436.145,E2 -436.145} C_VEL
LIN {X 0,Y 760.454,Z 641.677,A -85,B 0,C 180,E1 -438.713,E2 -438.713} C_VEL
LIN {X 0,Y 760.433,Z 649.485,A -85,B 0,C 180,E1 -439.619,E2 -439.619} C_VEL
LIN {X 0,Y 760.468,Z 754.939,A -85,B 0,C 180,E1 -440.624,E2 -440.624} C_VEL
LIN {X 0,Y 760.442,Z 764.938,A -85,B 0,C 180,E1 -440.774,E2 -440.774} C_VEL
LIN {X 0,Y 760.475,Z 776.182,A -85,B 0,C 180,E1 -441.025,E2 -441.025} C_VEL
LIN {X 0,Y 760.5,Z 786.28,A -85,B 0,C 180,E1 -441.326,E2 -441.326} C_VEL
LIN {X 0,Y 760.485,Z 796.776,A -85,B 0,C 180,E1 -441.726,E2 -441.726} C_VEL
LIN {X 0,Y 760.468,Z 806.622,A -85,B 0,C 180,E1 -442.192,E2 -442.192} C_VEL
LIN {X 0,Y 760.473,Z 815.845,A -85,B 0,C 180,E1 -442.724,E2 -442.724} C_VEL
LIN {X 0,Y 760.464,Z 823.587,A -85,B 0,C 180,E1 -443.256,E2 -443.256} C_VEL
LIN {X 0,Y 760.452,Z 830.356,A -85,B 0,C 180,E1 -443.8,E2 -443.8} C_VEL
LIN {X 0,Y 760.446,Z 837.164,A -85,B 0,C 180,E1 -444.45,E2 -444.45} C_VEL
LIN {X 0,Y 760.44,Z 843.951,A -85,B 0,C 180,E1 -445.245,E2 -445.245} C_VEL
LIN {X 0,Y 760.449,Z 849.401,A -85,B 0,C 180,E1 -446.039,E2 -446.039} C_VEL
LIN {X 0,Y 760.421,Z 853.688,A -85,B 0,C 180,E1 -446.832,E2 -446.832} C_VEL
LIN {X 0,Y 760.421,Z 855.971,A -85,B 0,C 180,E1 -447.36,E2 -447.36} C_VEL
LIN {X 0,Y 760.432,Z 859.204,A -85,B 0,C 180,E1 -448.417,E2 -448.417} C_VEL
LIN {X 0,Y 760.437,Z 860.715,A -85,B 0,C 180,E1 -449.472,E2 -449.472} C_VEL
LIN {X 0,Y 760.435,Z 861,A -85,B 0,C 180,E1 -450,E2 -450} C_VEL
LIN {X 0,Y 760.441,Z 860.14,A -85,B 0,C 180,E1 -451.056,E2 -451.056} C_VEL
LIN {X 0,Y 760.433,Z 859.204,A -85,B 0,C 180,E1 -451.584,E2 -451.584} C_VEL
LIN {X 0,Y 760.421,Z 855.97,A -85,B 0,C 180,E1 -452.64,E2 -452.64} C_VEL
LIN {X 0,Y 760.423,Z 852.421,A -85,B 0,C 180,E1 -453.433,E2 -453.433} C_VEL
LIN {X 0,Y 760.435,Z 847.766,A -85,B 0,C 180,E1 -454.226,E2 -454.226} C_VEL
LIN {X 0,Y 760.449,Z 841.855,A -85,B 0,C 180,E1 -455.02,E2 -455.02} C_VEL
LIN {X 0,Y 760.438,Z 834.463,A -85,B 0,C 180,E1 -455.815,E2 -455.815} C_VEL
LIN {X 0,Y 760.46,Z 826.971,A -85,B 0,C 180,E1 -456.479,E2 -456.479} C_VEL
LIN {X 0,Y 760.474,Z 819.883,A -85,B 0,C 180,E1 -457.01,E2 -457.01} C_VEL
LIN {X 0,Y 760.484,Z 811.473,A -85,B 0,C 180,E1 -457.542,E2 -457.542} C_VEL
LIN {X 0,Y 760.473,Z 802.697,A -85,B 0,C 180,E1 -458.008,E2 -458.008} C_VEL
LIN {X 0,Y 760.473,Z 791.819,A -85,B 0,C 180,E1 -458.475,E2 -458.475} C_VEL
LIN {X 0,Y 760.469,Z 780.97,A -85,B 0,C 180,E1 -458.842,E2 -458.842} C_VEL
LIN {X 0,Y 760.467,Z 769.892,A -85,B 0,C 180,E1 -459.126,E2 -459.126} C_VEL
LIN {X 0,Y 760.45,Z 758.808,A -85,B 0,C 180,E1 -459.326,E2 -459.326} C_VEL
LIN {X 0,Y 760.456,Z 740.223,A -85,B 0,C 180,E1 -459.527,E2 -459.527} C_VEL
LIN {X 0,Y 760.433,Z 649.483,A -85,B 0,C 180,E1 -460.381,E2 -460.381} C_VEL
LIN {X 0,Y 760.481,Z 627.793,A -85,B 0,C 180,E1 -462.906,E2 -462.906} C_VEL
LIN {X 0,Y 760.458,Z 606.97,A -85,B 0,C 180,E1 -465.356,E2 -465.356} C_VEL
LIN {X 0,Y 760.523,Z 584.99,A -85,B 0,C 180,E1 -467.971,E2 -467.971} C_VEL
LIN {X 0,Y 760.486,Z 564.167,A -85,B 0,C 180,E1 -470.487,E2 -470.487} C_VEL
LIN {X 0,Y 760.381,Z 562.697,A -85,B 0,C 180,E1 -470.702,E2 -470.702} C_VEL
LIN {X 0,Y 760.371,Z 562.695,A -85,B 0,C 180,E1 -472.9,E2 -472.9} C_VEL
LIN {X 0,Y 760.374,Z 562.695,A -85,B 0,C 180,E1 -475.071,E2 -475.071} C_VEL
LIN {X 0,Y 760.429,Z 562.693,A -85,B 0,C 180,E1 -477.423,E2 -477.423} C_VEL
LIN {X 0,Y 760.458,Z 562.692,A -85,B 0,C 180,E1 -480.024,E2 -480.024} C_VEL
LIN {X 0,Y 760.423,Z 562.691,A -85,B 0,C 180,E1 -482.293,E2 -482.293} C_VEL
LIN {X 0,Y 760.44,Z 562.689,A -85,B 0,C 180,E1 -484.186,E2 -484.186} C_VEL
LIN {X 0,Y 760.428,Z 562.688,A -85,B 0,C 180,E1 -486.739,E2 -486.739} C_VEL
LIN {X 0,Y 760.435,Z 562.688,A -85,B 0,C 180,E1 -488.782,E2 -488.782} C_VEL
LIN {X 0,Y 760.439,Z 562.69,A -85,B 0,C 180,E1 -490.948,E2 -490.948} C_VEL
LIN {X 0,Y 760.467,Z 562.689,A -85,B 0,C 180,E1 -493.694,E2 -493.694} C_VEL
LIN {X 0,Y 760.453,Z 562.685,A -85,B 0,C 180,E1 -496.305,E2 -496.305} C_VEL
LIN {X 0,Y 760.453,Z 562.686,A -85,B 0,C 180,E1 -498.457,E2 -498.457} C_VEL
LIN {X 0,Y 760.462,Z 562.688,A -85,B 0,C 180,E1 -500.688,E2 -500.688} C_VEL
LIN {X 0,Y 760.447,Z 562.694,A -85,B 0,C 180,E1 -503.26,E2 -503.26} C_VEL
LIN {X 0,Y 760.453,Z 562.685,A -85,B 0,C 180,E1 -505.815,E2 -505.815} C_VEL
LIN {X 0,Y 760.467,Z 562.686,A -85,B 0,C 180,E1 -508.331,E2 -508.331} C_VEL
LIN {X 0,Y 760.444,Z 562.699,A -85,B 0,C 180,E1 -510.779,E2 -510.779} C_VEL
LIN {X 0,Y 760.437,Z 562.691,A -85,B 0,C 180,E1 -513.17,E2 -513.17} C_VEL
LIN {X 0,Y 760.441,Z 562.687,A -85,B 0,C 180,E1 -515.512,E2 -515.512} C_VEL
LIN {X 0,Y 760.476,Z 562.683,A -85,B 0,C 180,E1 -517.813,E2 -517.813} C_VEL
LIN {X 0,Y 760.486,Z 562.685,A -85,B 0,C 180,E1 -520.075,E2 -520.075} C_VEL
LIN {X 0,Y 760.469,Z 562.693,A -85,B 0,C 180,E1 -522.305,E2 -522.305} C_VEL
LIN {X 0,Y 760.449,Z 562.696,A -85,B 0,C 180,E1 -524.507,E2 -524.507} C_VEL
LIN {X 0,Y 760.417,Z 562.695,A -85,B 0,C 180,E1 -526.686,E2 -526.686} C_VEL
LIN {X 0,Y 760.441,Z 562.699,A -85,B 0,C 180,E1 -528.308,E2 -528.308} C_VEL
LIN {X 0,Y 760.423,Z 562.696,A -85,B 0,C 180,E1 -530.456,E2 -530.456} C_VEL
LIN {X 0,Y 760.499,Z 562.865,A -85,B 0,C 180,E1 -531.659,E2 -531.659} C_VEL
LIN {X 0,Y 760.479,Z 582.088,A -85,B 0,C 180,E1 -534.361,E2 -534.361} C_VEL
LIN {X 0,Y 760.45,Z 599.897,A -85,B 0,C 180,E1 -536.832,E2 -536.832} C_VEL
LIN {X 0,Y 760.474,Z 617.188,A -85,B 0,C 180,E1 -539.208,E2 -539.208} C_VEL
LIN {X 0,Y 760.466,Z 620.566,A -85,B 0,C 180,E1 -539.67,E2 -539.67} C_VEL
LIN {X 0,Y 760.467,Z 725.515,A -85,B 0,C 180,E1 -540.676,E2 -540.676} C_VEL
LIN {X 0,Y 760.46,Z 735.214,A -85,B 0,C 180,E1 -540.824,E2 -540.824} C_VEL
LIN {X 0,Y 760.474,Z 745.667,A -85,B 0,C 180,E1 -541.055,E2 -541.055} C_VEL
LIN {X 0,Y 760.481,Z 756.7,A -85,B 0,C 180,E1 -541.385,E2 -541.385} C_VEL
LIN {X 0,Y 760.47,Z 767.019,A -85,B 0,C 180,E1 -541.781,E2 -541.781} C_VEL
LIN {X 0,Y 760.464,Z 776.746,A -85,B 0,C 180,E1 -542.243,E2 -542.243} C_VEL
LIN {X 0,Y 760.461,Z 785.885,A -85,B 0,C 180,E1 -542.772,E2 -542.772} C_VEL
LIN {X 0,Y 760.456,Z 793.583,A -85,B 0,C 180,E1 -543.3,E2 -543.3} C_VEL
LIN {X 0,Y 760.451,Z 801.596,A -85,B 0,C 180,E1 -543.961,E2 -543.961} C_VEL
LIN {X 0,Y 760.444,Z 808.297,A -85,B 0,C 180,E1 -544.623,E2 -544.623} C_VEL
LIN {X 0,Y 760.43,Z 813.918,A -85,B 0,C 180,E1 -545.285,E2 -545.285} C_VEL
LIN {X 0,Y 760.445,Z 819.232,A -85,B 0,C 180,E1 -546.054,E2 -546.054} C_VEL
LIN {X 0,Y 760.435,Z 823.691,A -85,B 0,C 180,E1 -546.877,E2 -546.877} C_VEL
LIN {X 0,Y 760.455,Z 825.987,A -85,B 0,C 180,E1 -547.409,E2 -547.409} C_VEL
LIN {X 0,Y 760.425,Z 827.957,A -85,B 0,C 180,E1 -548.016,E2 -548.016} C_VEL
LIN {X 0,Y 759.737,Z 829.189,A -85,B 0,C 180,E1 -548.451,E2 -548.451} C_VEL
LIN {X 0,Y 756.855,Z 830.449,A -85,B 0,C 180,E1 -549.161,E2 -549.161} C_VEL
LIN {X 0,Y 754.435,Z 830.935,A -85,B 0,C 180,E1 -549.736,E2 -549.736} C_VEL
LIN {X 0,Y 753.398,Z 830.954,A -85,B 0,C 180,E1 -550.179,E2 -550.179} C_VEL
LIN {X 0,Y 753.315,Z 830.867,A -85,B 0,C 180,E1 -550.329,E2 -550.329} C_VEL
LIN {X 0,Y 753.327,Z 829.887,A -85,B 0,C 180,E1 -551.26,E2 -551.26} C_VEL
LIN {X 0,Y 753.348,Z 828.84,A -85,B 0,C 180,E1 -551.803,E2 -551.803} C_VEL
LIN {X 0,Y 753.333,Z 826.756,A -85,B 0,C 180,E1 -552.503,E2 -552.503} C_VEL
LIN {X 0,Y 753.345,Z 822.796,A -85,B 0,C 180,E1 -553.441,E2 -553.441} C_VEL
LIN {X 0,Y 753.355,Z 818.096,A -85,B 0,C 180,E1 -554.264,E2 -554.264} C_VEL
LIN {X 0,Y 753.352,Z 812.067,A -85,B 0,C 180,E1 -555.09,E2 -555.09} C_VEL
LIN {X 0,Y 753.385,Z 804.439,A -85,B 0,C 180,E1 -555.918,E2 -555.918} C_VEL
LIN {X 0,Y 753.38,Z 797.151,A -85,B 0,C 180,E1 -556.572,E2 -556.572} C_VEL
LIN {X 0,Y 753.424,Z 789.192,A -85,B 0,C 180,E1 -557.168,E2 -557.168} C_VEL
LIN {X 0,Y 753.415,Z 780.263,A -85,B 0,C 180,E1 -557.726,E2 -557.726} C_VEL
LIN {X 0,Y 753.451,Z 770.796,A -85,B 0,C 180,E1 -558.215,E2 -558.215} C_VEL
LIN {X 0,Y 753.468,Z 762.46,A -85,B 0,C 180,E1 -558.577,E2 -558.577} C_VEL
LIN {X 0,Y 753.464,Z 751.576,A -85,B 0,C 180,E1 -558.953,E2 -558.953} C_VEL
LIN {X 0,Y 753.451,Z 740.139,A -85,B 0,C 180,E1 -559.252,E2 -559.252} C_VEL
LIN {X 0,Y 753.513,Z 728.54,A -85,B 0,C 180,E1 -559.462,E2 -559.462} C_VEL
LIN {X 0,Y 753.522,Z 708.764,A -85,B 0,C 180,E1 -559.674,E2 -559.674} C_VEL
LIN {X 0,Y 753.382,Z 620.724,A -85,B 0,C 180,E1 -560.511,E2 -560.511} C_VEL
LIN {X 0,Y 753.391,Z 603.808,A -85,B 0,C 180,E1 -562.84,E2 -562.84} C_VEL
LIN {X 0,Y 753.43,Z 587.125,A -85,B 0,C 180,E1 -565.171,E2 -565.171} C_VEL
LIN {X 0,Y 753.473,Z 569.249,A -85,B 0,C 180,E1 -567.698,E2 -567.698} C_VEL
LIN {X 0,Y 753.41,Z 563.566,A -85,B 0,C 180,E1 -568.531,E2 -568.531} C_VEL
LIN {X 0,Y 753.394,Z 563.564,A -85,B 0,C 180,E1 -570.753,E2 -570.753} C_VEL
LIN {X 0,Y 753.415,Z 563.562,A -85,B 0,C 180,E1 -573.204,E2 -573.204} C_VEL
LIN {X 0,Y 753.405,Z 563.574,A -85,B 0,C 180,E1 -575.853,E2 -575.853} C_VEL
LIN {X 0,Y 753.419,Z 563.572,A -85,B 0,C 180,E1 -577.849,E2 -577.849} C_VEL
LIN {X 0,Y 753.403,Z 563.568,A -85,B 0,C 180,E1 -580.327,E2 -580.327} C_VEL
LIN {X 0,Y 753.406,Z 563.563,A -85,B 0,C 180,E1 -582.74,E2 -582.74} C_VEL
LIN {X 0,Y 753.417,Z 563.561,A -85,B 0,C 180,E1 -585.044,E2 -585.044} C_VEL
LIN {X 0,Y 753.423,Z 563.561,A -85,B 0,C 180,E1 -587.26,E2 -587.26} C_VEL
LIN {X 0,Y 753.411,Z 563.569,A -85,B 0,C 180,E1 -589.671,E2 -589.671} C_VEL
LIN {X 0,Y 753.413,Z 563.569,A -85,B 0,C 180,E1 -592.207,E2 -592.207} C_VEL
LIN {X 0,Y 753.408,Z 563.562,A -85,B 0,C 180,E1 -594.898,E2 -594.898} C_VEL
LIN {X 0,Y 753.419,Z 563.563,A -85,B 0,C 180,E1 -597.369,E2 -597.369} C_VEL
LIN {X 0,Y 753.411,Z 563.573,A -85,B 0,C 180,E1 -599.865,E2 -599.865} C_VEL
LIN {X 0,Y 753.412,Z 563.567,A -85,B 0,C 180,E1 -602.299,E2 -602.299} C_VEL
LIN {X 0,Y 753.397,Z 563.564,A -85,B 0,C 180,E1 -604.68,E2 -604.68} C_VEL
LIN {X 0,Y 753.42,Z 563.56,A -85,B 0,C 180,E1 -607.016,E2 -607.016} C_VEL
LIN {X 0,Y 753.421,Z 563.562,A -85,B 0,C 180,E1 -609.312,E2 -609.312} C_VEL
LIN {X 0,Y 753.404,Z 563.568,A -85,B 0,C 180,E1 -611.573,E2 -611.573} C_VEL
LIN {X 0,Y 753.402,Z 563.573,A -85,B 0,C 180,E1 -613.805,E2 -613.805} C_VEL
LIN {X 0,Y 753.392,Z 563.576,A -85,B 0,C 180,E1 -616.011,E2 -616.011} C_VEL
LIN {X 0,Y 753.408,Z 563.57,A -85,B 0,C 180,E1 -618.198,E2 -618.198} C_VEL
LIN {X 0,Y 753.41,Z 563.566,A -85,B 0,C 180,E1 -620.366,E2 -620.366} C_VEL
LIN {X 0,Y 753.414,Z 563.564,A -85,B 0,C 180,E1 -622.521,E2 -622.521} C_VEL
LIN {X 0,Y 753.432,Z 563.56,A -85,B 0,C 180,E1 -625.2,E2 -625.2} C_VEL
LIN {X 0,Y 753.439,Z 563.57,A -85,B 0,C 180,E1 -627.869,E2 -627.869} C_VEL
LIN {X 0,Y 753.426,Z 563.562,A -85,B 0,C 180,E1 -630.533,E2 -630.533} C_VEL
LIN {X 0,Y 753.409,Z 563.563,A -85,B 0,C 180,E1 -632.664,E2 -632.664} C_VEL
LIN {X 0,Y 753.432,Z 563.559,A -85,B 0,C 180,E1 -634.799,E2 -634.799} C_VEL
LIN {X 0,Y 753.413,Z 563.565,A -85,B 0,C 180,E1 -637.479,E2 -637.479} C_VEL
LIN {X 0,Y 753.433,Z 563.567,A -85,B 0,C 180,E1 -640.174,E2 -640.174} C_VEL
LIN {X 0,Y 753.418,Z 563.563,A -85,B 0,C 180,E1 -642.535,E2 -642.535} C_VEL
LIN {X 0,Y 753.406,Z 563.562,A -85,B 0,C 180,E1 -645.089,E2 -645.089} C_VEL
LIN {X 0,Y 753.412,Z 563.563,A -85,B 0,C 180,E1 -647.308,E2 -647.308} C_VEL
LIN {X 0,Y 753.405,Z 563.567,A -85,B 0,C 180,E1 -649.554,E2 -649.554} C_VEL
LIN {X 0,Y 753.41,Z 563.573,A -85,B 0,C 180,E1 -651.832,E2 -651.832} C_VEL
LIN {X 0,Y 753.408,Z 563.567,A -85,B 0,C 180,E1 -654.342,E2 -654.342} C_VEL
LIN {X 0,Y 753.432,Z 563.559,A -85,B 0,C 180,E1 -656.814,E2 -656.814} C_VEL
LIN {X 0,Y 753.431,Z 563.559,A -85,B 0,C 180,E1 -659.087,E2 -659.087} C_VEL
LIN {X 0,Y 753.403,Z 563.565,A -85,B 0,C 180,E1 -661.375,E2 -661.375} C_VEL
LIN {X 0,Y 753.416,Z 563.562,A -85,B 0,C 180,E1 -663.265,E2 -663.265} C_VEL
LIN {X 0,Y 753.396,Z 563.575,A -85,B 0,C 180,E1 -665.854,E2 -665.854} C_VEL
LIN {X 0,Y 753.413,Z 563.573,A -85,B 0,C 180,E1 -667.85,E2 -667.85} C_VEL
LIN {X 0,Y 753.41,Z 563.567,A -85,B 0,C 180,E1 -670.329,E2 -670.329} C_VEL
LIN {X 0,Y 753.421,Z 563.561,A -85,B 0,C 180,E1 -672.74,E2 -672.74} C_VEL
LIN {X 0,Y 753.412,Z 563.561,A -85,B 0,C 180,E1 -675.044,E2 -675.044} C_VEL
LIN {X 0,Y 753.404,Z 563.564,A -85,B 0,C 180,E1 -677.262,E2 -677.262} C_VEL
LIN {X 0,Y 753.403,Z 563.57,A -85,B 0,C 180,E1 -679.673,E2 -679.673} C_VEL
LIN {X 0,Y 753.42,Z 563.568,A -85,B 0,C 180,E1 -682.207,E2 -682.207} C_VEL
LIN {X 0,Y 753.404,Z 563.562,A -85,B 0,C 180,E1 -684.899,E2 -684.899} C_VEL
LIN {X 0,Y 753.4,Z 563.565,A -85,B 0,C 180,E1 -687.369,E2 -687.369} C_VEL
LIN {X 0,Y 753.413,Z 563.573,A -85,B 0,C 180,E1 -689.866,E2 -689.866} C_VEL
LIN {X 0,Y 753.42,Z 563.566,A -85,B 0,C 180,E1 -692.3,E2 -692.3} C_VEL
LIN {X 0,Y 753.418,Z 563.561,A -85,B 0,C 180,E1 -694.681,E2 -694.681} C_VEL
LIN {X 0,Y 753.382,Z 563.565,A -85,B 0,C 180,E1 -697.015,E2 -697.015} C_VEL
LIN {X 0,Y 753.404,Z 563.564,A -85,B 0,C 180,E1 -699.312,E2 -699.312} C_VEL
LIN {X 0,Y 753.387,Z 563.57,A -85,B 0,C 180,E1 -701.573,E2 -701.573} C_VEL
LIN {X 0,Y 753.392,Z 563.574,A -85,B 0,C 180,E1 -703.805,E2 -703.805} C_VEL
LIN {X 0,Y 753.415,Z 563.573,A -85,B 0,C 180,E1 -706.012,E2 -706.012} C_VEL
LIN {X 0,Y 753.419,Z 563.568,A -85,B 0,C 180,E1 -708.198,E2 -708.198} C_VEL
LIN {X 0,Y 753.426,Z 563.564,A -85,B 0,C 180,E1 -710.367,E2 -710.367} C_VEL
LIN {X 0,Y 753.423,Z 563.562,A -85,B 0,C 180,E1 -712.522,E2 -712.522} C_VEL
LIN {X 0,Y 753.4,Z 563.564,A -85,B 0,C 180,E1 -714.666,E2 -714.666} C_VEL
LIN {X 0,Y 753.379,Z 563.565,A -85,B 0,C 180,E1 -716.802,E2 -716.802} C_VEL
LIN {X 0,Y 753.395,Z 563.563,A -85,B 0,C 180,E1 -718.935,E2 -718.935} C_VEL
LIN {X 0,Y 753.389,Z 563.564,A -85,B 0,C 180,E1 -721.066,E2 -721.066} C_VEL
LIN {X 0,Y 753.361,Z 563.568,A -85,B 0,C 180,E1 -723.198,E2 -723.198} C_VEL
LIN {X 0,Y 753.414,Z 563.561,A -85,B 0,C 180,E1 -724.8,E2 -724.8} C_VEL
LIN {X 0,Y 753.381,Z 563.565,A -85,B 0,C 180,E1 -726.942,E2 -726.942} C_VEL
LIN {X 0,Y 753.384,Z 563.565,A -85,B 0,C 180,E1 -729.094,E2 -729.094} C_VEL
LIN {X 0,Y 753.364,Z 563.569,A -85,B 0,C 180,E1 -731.259,E2 -731.259} C_VEL
LIN {X 0,Y 753.397,Z 563.563,A -85,B 0,C 180,E1 -732.893,E2 -732.893} C_VEL
LIN {X 0,Y 753.389,Z 563.564,A -85,B 0,C 180,E1 -735.089,E2 -735.089} C_VEL
LIN {X 0,Y 753.387,Z 563.566,A -85,B 0,C 180,E1 -737.308,E2 -737.308} C_VEL
LIN {X 0,Y 753.385,Z 563.57,A -85,B 0,C 180,E1 -739.555,E2 -739.555} C_VEL
LIN {X 0,Y 753.393,Z 563.575,A -85,B 0,C 180,E1 -741.832,E2 -741.832} C_VEL
LIN {X 0,Y 753.407,Z 563.567,A -85,B 0,C 180,E1 -744.341,E2 -744.341} C_VEL
LIN {X 0,Y 753.392,Z 563.564,A -85,B 0,C 180,E1 -746.807,E2 -746.807} C_VEL
LIN {X 0,Y 753.37,Z 563.567,A -85,B 0,C 180,E1 -749.077,E2 -749.077} C_VEL
LIN {X 0,Y 753.377,Z 563.568,A -85,B 0,C 180,E1 -751.376,E2 -751.376} C_VEL
LIN {X 0,Y 753.396,Z 563.577,A -85,B 0,C 180,E1 -753.906,E2 -753.906} C_VEL
LIN {X 0,Y 753.382,Z 563.567,A -85,B 0,C 180,E1 -756.515,E2 -756.515} C_VEL
LIN {X 0,Y 753.389,Z 563.565,A -85,B 0,C 180,E1 -758.651,E2 -758.651} C_VEL
LIN {X 0,Y 753.386,Z 563.565,A -85,B 0,C 180,E1 -761.142,E2 -761.142} C_VEL
LIN {X 0,Y 753.397,Z 563.568,A -85,B 0,C 180,E1 -763.516,E2 -763.516} C_VEL
LIN {X 0,Y 753.378,Z 563.576,A -85,B 0,C 180,E1 -765.789,E2 -765.789} C_VEL
LIN {X 0,Y 753.39,Z 563.575,A -85,B 0,C 180,E1 -768.054,E2 -768.054} C_VEL
LIN {X 0,Y 753.387,Z 563.567,A -85,B 0,C 180,E1 -770.504,E2 -770.504} C_VEL
LIN {X 0,Y 753.346,Z 563.57,A -85,B 0,C 180,E1 -772.818,E2 -772.818} C_VEL
LIN {X 0,Y 753.35,Z 563.569,A -85,B 0,C 180,E1 -774.905,E2 -774.905} C_VEL
LIN {X 0,Y 753.364,Z 563.567,A -85,B 0,C 180,E1 -776.801,E2 -776.801} C_VEL
LIN {X 0,Y 753.36,Z 563.568,A -85,B 0,C 180,E1 -778.801,E2 -778.801} C_VEL
LIN {X 0,Y 753.357,Z 563.568,A -85,B 0,C 180,E1 -780.924,E2 -780.924} C_VEL
LIN {X 0,Y 753.372,Z 563.567,A -85,B 0,C 180,E1 -783.196,E2 -783.196} C_VEL
LIN {X 0,Y 753.338,Z 563.572,A -85,B 0,C 180,E1 -785.266,E2 -785.266} C_VEL
LIN {X 0,Y 753.376,Z 563.572,A -85,B 0,C 180,E1 -787.592,E2 -787.592} C_VEL
LIN {X 0,Y 753.355,Z 563.591,A -85,B 0,C 180,E1 -789.239,E2 -789.239} C_VEL
LIN {X 0,Y 753.528,Z 573.424,A -85,B 0,C 180,E1 -790.449,E2 -790.449} C_VEL
LIN {X 0,Y 753.496,Z 593.205,A -85,B 0,C 180,E1 -792.848,E2 -792.848} C_VEL
LIN {X 0,Y 753.445,Z 613.737,A -85,B 0,C 180,E1 -795.304,E2 -795.304} C_VEL
LIN {X 0,Y 753.433,Z 635.892,A -85,B 0,C 180,E1 -797.926,E2 -797.926} C_VEL
LIN {X 0,Y 753.366,Z 649.485,A -85,B 0,C 180,E1 -799.521,E2 -799.521} C_VEL
LIN {X 0,Y 753.472,Z 754.938,A -85,B 0,C 180,E1 -800.536,E2 -800.536} C_VEL
LIN {X 0,Y 753.453,Z 764.94,A -85,B 0,C 180,E1 -800.688,E2 -800.688} C_VEL
LIN {X 0,Y 753.447,Z 776.184,A -85,B 0,C 180,E1 -800.941,E2 -800.941} C_VEL
LIN {X 0,Y 753.476,Z 786.284,A -85,B 0,C 180,E1 -801.244,E2 -801.244} C_VEL
LIN {X 0,Y 753.455,Z 796.779,A -85,B 0,C 180,E1 -801.648,E2 -801.648} C_VEL
LIN {X 0,Y 753.434,Z 806.625,A -85,B 0,C 180,E1 -802.119,E2 -802.119} C_VEL
LIN {X 0,Y 753.418,Z 815.847,A -85,B 0,C 180,E1 -802.656,E2 -802.656} C_VEL
LIN {X 0,Y 753.389,Z 823.587,A -85,B 0,C 180,E1 -803.192,E2 -803.192} C_VEL
LIN {X 0,Y 753.373,Z 831.631,A -85,B 0,C 180,E1 -803.862,E2 -803.862} C_VEL
LIN {X 0,Y 753.371,Z 838.163,A -85,B 0,C 180,E1 -804.512,E2 -804.512} C_VEL
LIN {X 0,Y 753.358,Z 843.952,A -85,B 0,C 180,E1 -805.2,E2 -805.2} C_VEL
LIN {X 0,Y 753.37,Z 849.402,A -85,B 0,C 180,E1 -806.002,E2 -806.002} C_VEL
LIN {X 0,Y 753.351,Z 853.689,A -85,B 0,C 180,E1 -806.802,E2 -806.802} C_VEL
LIN {X 0,Y 753.331,Z 855.972,A -85,B 0,C 180,E1 -807.335,E2 -807.335} C_VEL
LIN {X 0,Y 753.332,Z 859.203,A -85,B 0,C 180,E1 -808.402,E2 -808.402} C_VEL
LIN {X 0,Y 753.338,Z 860.715,A -85,B 0,C 180,E1 -809.467,E2 -809.467} C_VEL
LIN {X 0,Y 753.335,Z 861,A -85,B 0,C 180,E1 -810,E2 -810} C_VEL
LIN {X 0,Y 753.341,Z 860.141,A -85,B 0,C 180,E1 -811.066,E2 -811.066} C_VEL
LIN {X 0,Y 753.332,Z 859.203,A -85,B 0,C 180,E1 -811.599,E2 -811.599} C_VEL
LIN {X 0,Y 753.331,Z 855.971,A -85,B 0,C 180,E1 -812.665,E2 -812.665} C_VEL
LIN {X 0,Y 753.328,Z 852.422,A -85,B 0,C 180,E1 -813.465,E2 -813.465} C_VEL
LIN {X 0,Y 753.34,Z 847.766,A -85,B 0,C 180,E1 -814.266,E2 -814.266} C_VEL
LIN {X 0,Y 753.371,Z 841.855,A -85,B 0,C 180,E1 -815.067,E2 -815.067} C_VEL
LIN {X 0,Y 753.355,Z 835.007,A -85,B 0,C 180,E1 -815.819,E2 -815.819} C_VEL
LIN {X 0,Y 753.401,Z 826.97,A -85,B 0,C 180,E1 -816.54,E2 -816.54} C_VEL
LIN {X 0,Y 753.423,Z 819.885,A -85,B 0,C 180,E1 -817.076,E2 -817.076} C_VEL
LIN {X 0,Y 753.422,Z 811.476,A -85,B 0,C 180,E1 -817.613,E2 -817.613} C_VEL
LIN {X 0,Y 753.442,Z 801.219,A -85,B 0,C 180,E1 -818.151,E2 -818.151} C_VEL
LIN {X 0,Y 753.441,Z 791.823,A -85,B 0,C 180,E1 -818.554,E2 -818.554} C_VEL
LIN {X 0,Y 753.446,Z 780.972,A -85,B 0,C 180,E1 -818.925,E2 -818.925} C_VEL
LIN {X 0,Y 753.443,Z 769.892,A -85,B 0,C 180,E1 -819.211,E2 -819.211} C_VEL
LIN {X 0,Y 753.468,Z 758.808,A -85,B 0,C 180,E1 -819.413,E2 -819.413} C_VEL
LIN {X 0,Y 753.471,Z 740.223,A -85,B 0,C 180,E1 -819.616,E2 -819.616} C_VEL
LIN {X 0,Y 753.367,Z 649.483,A -85,B 0,C 180,E1 -820.48,E2 -820.48} C_VEL
LIN {X 0,Y 753.438,Z 628.95,A -85,B 0,C 180,E1 -822.892,E2 -822.892} C_VEL
LIN {X 0,Y 753.432,Z 609.284,A -85,B 0,C 180,E1 -825.226,E2 -825.226} C_VEL
LIN {X 0,Y 753.491,Z 588.461,A -85,B 0,C 180,E1 -827.725,E2 -827.725} C_VEL
LIN {X 0,Y 753.558,Z 568.538,A -85,B 0,C 180,E1 -830.147,E2 -830.147} C_VEL
LIN {X 0,Y 753.362,Z 563.573,A -85,B 0,C 180,E1 -830.779,E2 -830.779} C_VEL
LIN {X 0,Y 753.331,Z 563.573,A -85,B 0,C 180,E1 -833.001,E2 -833.001} C_VEL
LIN {X 0,Y 753.336,Z 563.572,A -85,B 0,C 180,E1 -834.734,E2 -834.734} C_VEL
LIN {X 0,Y 753.371,Z 563.568,A -85,B 0,C 180,E1 -836.804,E2 -836.804} C_VEL
LIN {X 0,Y 753.362,Z 563.57,A -85,B 0,C 180,E1 -839.077,E2 -839.077} C_VEL
LIN {X 0,Y 753.381,Z 563.572,A -85,B 0,C 180,E1 -841.376,E2 -841.376} C_VEL
LIN {X 0,Y 753.41,Z 563.57,A -85,B 0,C 180,E1 -843.905,E2 -843.905} C_VEL
LIN {X 0,Y 753.378,Z 563.566,A -85,B 0,C 180,E1 -846.515,E2 -846.515} C_VEL
LIN {X 0,Y 753.389,Z 563.565,A -85,B 0,C 180,E1 -848.651,E2 -848.651} C_VEL
LIN {X 0,Y 753.422,Z 563.571,A -85,B 0,C 180,E1 -851.306,E2 -851.306} C_VEL
LIN {X 0,Y 753.416,Z 563.571,A -85,B 0,C 180,E1 -853.518,E2 -853.518} C_VEL
LIN {X 0,Y 753.402,Z 563.566,A -85,B 0,C 180,E1 -855.791,E2 -855.791} C_VEL
LIN {X 0,Y 753.399,Z 563.564,A -85,B 0,C 180,E1 -858.054,E2 -858.054} C_VEL
LIN {X 0,Y 753.412,Z 563.564,A -85,B 0,C 180,E1 -860.502,E2 -860.502} C_VEL
LIN {X 0,Y 753.409,Z 563.575,A -85,B 0,C 180,E1 -863.087,E2 -863.087} C_VEL
LIN {X 0,Y 753.423,Z 563.561,A -85,B 0,C 180,E1 -865.835,E2 -865.835} C_VEL
LIN {X 0,Y 753.426,Z 563.56,A -85,B 0,C 180,E1 -868,E2 -868} C_VEL
LIN {X 0,Y 753.417,Z 563.568,A -85,B 0,C 180,E1 -870.479,E2 -870.479} C_VEL
LIN {X 0,Y 753.397,Z 563.573,A -85,B 0,C 180,E1 -872.899,E2 -872.899} C_VEL
LIN {X 0,Y 753.411,Z 563.576,A -85,B 0,C 180,E1 -874.681,E2 -874.681} C_VEL
LIN {X 0,Y 753.384,Z 563.57,A -85,B 0,C 180,E1 -877.015,E2 -877.015} C_VEL
LIN {X 0,Y 753.412,Z 563.563,A -85,B 0,C 180,E1 -879.312,E2 -879.312} C_VEL
LIN {X 0,Y 753.413,Z 563.562,A -85,B 0,C 180,E1 -881.573,E2 -881.573} C_VEL
LIN {X 0,Y 753.408,Z 563.565,A -85,B 0,C 180,E1 -883.805,E2 -883.805} C_VEL
LIN {X 0,Y 753.405,Z 563.57,A -85,B 0,C 180,E1 -886.012,E2 -886.012} C_VEL
LIN {X 0,Y 753.41,Z 563.575,A -85,B 0,C 180,E1 -888.198,E2 -888.198} C_VEL
LIN {X 0,Y 753.399,Z 563.574,A -85,B 0,C 180,E1 -890.366,E2 -890.366} C_VEL
LIN {X 0,Y 753.457,Z 563.679,A -85,B 0,C 180,E1 -891.597,E2 -891.597} C_VEL
LIN {X 0,Y 753.468,Z 581.519,A -85,B 0,C 180,E1 -894.131,E2 -894.131} C_VEL
LIN {X 0,Y 753.431,Z 598.671,A -85,B 0,C 180,E1 -896.535,E2 -896.535} C_VEL
LIN {X 0,Y 753.392,Z 615.952,A -85,B 0,C 180,E1 -898.934,E2 -898.934} C_VEL
LIN {X 0,Y 753.41,Z 620.532,A -85,B 0,C 180,E1 -899.567,E2 -899.567} C_VEL
LIN {X 0,Y 753.573,Z 643.728,A -85,B 0,C 180,E1 -899.8,E2 -899.8} C_VEL
LIN {X 0,Y 753.463,Z 725.122,A -85,B 0,C 180,E1 -900.582,E2 -900.582} C_VEL
LIN {X 0,Y 753.449,Z 735.785,A -85,B 0,C 180,E1 -900.749,E2 -900.749} C_VEL
LIN {X 0,Y 753.448,Z 746.676,A -85,B 0,C 180,E1 -900.999,E2 -900.999} C_VEL
LIN {X 0,Y 753.466,Z 755.648,A -85,B 0,C 180,E1 -901.265,E2 -901.265} C_VEL
LIN {X 0,Y 753.438,Z 766.175,A -85,B 0,C 180,E1 -901.665,E2 -901.665} C_VEL
LIN {X 0,Y 753.409,Z 776.061,A -85,B 0,C 180,E1 -902.131,E2 -902.131} C_VEL
LIN {X 0,Y 753.393,Z 785.312,A -85,B 0,C 180,E1 -902.664,E2 -902.664} C_VEL
LIN {X 0,Y 753.383,Z 793.104,A -85,B 0,C 180,E1 -903.198,E2 -903.198} C_VEL
LIN {X 0,Y 753.365,Z 801.193,A -85,B 0,C 180,E1 -903.865,E2 -903.865} C_VEL
LIN {X 0,Y 753.353,Z 807.967,A -85,B 0,C 180,E1 -904.533,E2 -904.533} C_VEL
LIN {X 0,Y 753.37,Z 812.624,A -85,B 0,C 180,E1 -905.067,E2 -905.067} C_VEL
LIN {X 0,Y 753.348,Z 818.375,A -85,B 0,C 180,E1 -905.87,E2 -905.87} C_VEL
LIN {X 0,Y 753.34,Z 822.922,A -85,B 0,C 180,E1 -906.674,E2 -906.674} C_VEL
LIN {X 0,Y 753.35,Z 826.378,A -85,B 0,C 180,E1 -907.479,E2 -907.479} C_VEL
LIN {X 0,Y 753.324,Z 829.404,A -85,B 0,C 180,E1 -908.555,E2 -908.555} C_VEL
LIN {X 0,Y 753.345,Z 830.35,A -85,B 0,C 180,E1 -909.094,E2 -909.094} C_VEL
LIN {X 0,Y 753.319,Z 830.957,A -85,B 0,C 180,E1 -910.175,E2 -910.175} C_VEL
LIN {X 0,Y 753.315,Z 830.867,A -85,B 0,C 180,E1 -910.329,E2 -910.329} C_VEL
LIN {X 0,Y 752.644,Z 830.608,A -85,B 0,C 180,E1 -910.776,E2 -910.776} C_VEL
LIN {X 0,Y 749.768,Z 829.552,A -85,B 0,C 180,E1 -911.497,E2 -911.497} C_VEL
LIN {X 0,Y 747.349,Z 828.23,A -85,B 0,C 180,E1 -912.07,E2 -912.07} C_VEL
LIN {X 0,Y 746.316,Z 826.827,A -85,B 0,C 180,E1 -912.504,E2 -912.504} C_VEL
LIN {X 0,Y 746.236,Z 826.264,A -85,B 0,C 180,E1 -912.65,E2 -912.65} C_VEL
LIN {X 0,Y 746.251,Z 822.279,A -85,B 0,C 180,E1 -913.571,E2 -913.571} C_VEL
LIN {X 0,Y 746.265,Z 817.424,A -85,B 0,C 180,E1 -914.402,E2 -914.402} C_VEL
LIN {X 0,Y 746.29,Z 811.223,A -85,B 0,C 180,E1 -915.236,E2 -915.236} C_VEL
LIN {X 0,Y 746.301,Z 804.872,A -85,B 0,C 180,E1 -915.934,E2 -915.934} C_VEL
LIN {X 0,Y 746.308,Z 797.672,A -85,B 0,C 180,E1 -916.593,E2 -916.593} C_VEL
LIN {X 0,Y 746.352,Z 788.76,A -85,B 0,C 180,E1 -917.265,E2 -917.265} C_VEL
LIN {X 0,Y 746.386,Z 781.018,A -85,B 0,C 180,E1 -917.758,E2 -917.758} C_VEL
LIN {X 0,Y 746.425,Z 771.713,A -85,B 0,C 180,E1 -918.251,E2 -918.251} C_VEL
LIN {X 0,Y 746.44,Z 761.982,A -85,B 0,C 180,E1 -918.676,E2 -918.676} C_VEL
LIN {X 0,Y 746.461,Z 750.597,A -85,B 0,C 180,E1 -919.066,E2 -919.066} C_VEL
LIN {X 0,Y 746.461,Z 739.613,A -85,B 0,C 180,E1 -919.351,E2 -919.351} C_VEL
LIN {X 0,Y 746.508,Z 729.047,A -85,B 0,C 180,E1 -919.546,E2 -919.546} C_VEL
LIN {X 0,Y 746.546,Z 709.623,A -85,B 0,C 180,E1 -919.757,E2 -919.757} C_VEL
LIN {X 0,Y 746.4,Z 621.343,A -85,B 0,C 180,E1 -920.604,E2 -920.604} C_VEL
LIN {X 0,Y 746.312,Z 620.527,A -85,B 0,C 180,E1 -920.624,E2 -920.624} C_VEL
LIN {X 0,Y 746.333,Z 604.44,A -85,B 0,C 180,E1 -922.874,E2 -922.874} C_VEL
LIN {X 0,Y 746.404,Z 587.413,A -85,B 0,C 180,E1 -925.276,E2 -925.276} C_VEL
LIN {X 0,Y 746.457,Z 569.531,A -85,B 0,C 180,E1 -927.829,E2 -927.829} C_VEL
LIN {X 0,Y 746.353,Z 564.446,A -85,B 0,C 180,E1 -928.596,E2 -928.596} C_VEL
LIN {X 0,Y 746.349,Z 564.445,A -85,B 0,C 180,E1 -930.45,E2 -930.45} C_VEL
LIN {X 0,Y 746.366,Z 564.439,A -85,B 0,C 180,E1 -932.977,E2 -932.977} C_VEL
LIN {X 0,Y 746.374,Z 564.443,A -85,B 0,C 180,E1 -935.58,E2 -935.58} C_VEL
LIN {X 0,Y 746.36,Z 564.453,A -85,B 0,C 180,E1 -937.971,E2 -937.971} C_VEL
LIN {X 0,Y 746.375,Z 564.44,A -85,B 0,C 180,E1 -940.522,E2 -940.522} C_VEL
LIN {X 0,Y 746.353,Z 564.441,A -85,B 0,C 180,E1 -942.944,E2 -942.944} C_VEL
LIN {X 0,Y 746.367,Z 564.443,A -85,B 0,C 180,E1 -945.498,E2 -945.498} C_VEL
LIN {X 0,Y 746.352,Z 564.452,A -85,B 0,C 180,E1 -947.851,E2 -947.851} C_VEL
LIN {X 0,Y 746.365,Z 564.446,A -85,B 0,C 180,E1 -949.643,E2 -949.643} C_VEL
LIN {X 0,Y 746.359,Z 564.452,A -85,B 0,C 180,E1 -952.028,E2 -952.028} C_VEL
LIN {X 0,Y 746.369,Z 564.443,A -85,B 0,C 180,E1 -954.419,E2 -954.419} C_VEL
LIN {X 0,Y 746.373,Z 564.438,A -85,B 0,C 180,E1 -957.022,E2 -957.022} C_VEL
LIN {X 0,Y 746.364,Z 564.444,A -85,B 0,C 180,E1 -959.55,E2 -959.55} C_VEL
LIN {X 0,Y 746.381,Z 564.449,A -85,B 0,C 180,E1 -962.016,E2 -962.016} C_VEL
LIN {X 0,Y 746.383,Z 564.441,A -85,B 0,C 180,E1 -964.425,E2 -964.425} C_VEL
LIN {X 0,Y 746.363,Z 564.439,A -85,B 0,C 180,E1 -966.882,E2 -966.882} C_VEL
LIN {X 0,Y 746.372,Z 564.439,A -85,B 0,C 180,E1 -969.107,E2 -969.107} C_VEL
LIN {X 0,Y 746.391,Z 564.439,A -85,B 0,C 180,E1 -971.409,E2 -971.409} C_VEL
LIN {X 0,Y 746.381,Z 564.444,A -85,B 0,C 180,E1 -973.648,E2 -973.648} C_VEL
LIN {X 0,Y 746.35,Z 564.453,A -85,B 0,C 180,E1 -975.877,E2 -975.877} C_VEL
LIN {X 0,Y 746.38,Z 564.448,A -85,B 0,C 180,E1 -978.085,E2 -978.085} C_VEL
LIN {X 0,Y 746.365,Z 564.445,A -85,B 0,C 180,E1 -980.275,E2 -980.275} C_VEL
LIN {X 0,Y 746.376,Z 564.441,A -85,B 0,C 180,E1 -982.45,E2 -982.45} C_VEL
LIN {X 0,Y 746.403,Z 564.435,A -85,B 0,C 180,E1 -985.155,E2 -985.155} C_VEL
LIN {X 0,Y 746.402,Z 564.446,A -85,B 0,C 180,E1 -987.849,E2 -987.849} C_VEL
LIN {X 0,Y 746.381,Z 564.44,A -85,B 0,C 180,E1 -990.538,E2 -990.538} C_VEL
LIN {X 0,Y 746.363,Z 564.44,A -85,B 0,C 180,E1 -992.689,E2 -992.689} C_VEL
LIN {X 0,Y 746.403,Z 564.435,A -85,B 0,C 180,E1 -994.845,E2 -994.845} C_VEL
LIN {X 0,Y 746.376,Z 564.443,A -85,B 0,C 180,E1 -997.55,E2 -997.55} C_VEL
LIN {X 0,Y 746.367,Z 564.449,A -85,B 0,C 180,E1 -999.807,E2 -999.807} C_VEL
LIN {X 0,Y 746.378,Z 564.451,A -85,B 0,C 180,E1 -1001.915,E2 -1001.915} C_VEL
LIN {X 0,Y 746.38,Z 564.438,A -85,B 0,C 180,E1 -1004.678,E2 -1004.678} C_VEL
LIN {X 0,Y 746.407,Z 564.434,A -85,B 0,C 180,E1 -1006.912,E2 -1006.912} C_VEL
LIN {X 0,Y 746.369,Z 564.439,A -85,B 0,C 180,E1 -1009.176,E2 -1009.176} C_VEL
LIN {X 0,Y 746.379,Z 564.446,A -85,B 0,C 180,E1 -1011.711,E2 -1011.711} C_VEL
LIN {X 0,Y 746.377,Z 564.442,A -85,B 0,C 180,E1 -1014.388,E2 -1014.388} C_VEL
LIN {X 0,Y 746.395,Z 564.435,A -85,B 0,C 180,E1 -1016.937,E2 -1016.937} C_VEL
LIN {X 0,Y 746.388,Z 564.437,A -85,B 0,C 180,E1 -1019.221,E2 -1019.221} C_VEL
LIN {X 0,Y 746.372,Z 564.446,A -85,B 0,C 180,E1 -1021.705,E2 -1021.705} C_VEL
LIN {X 0,Y 746.38,Z 564.443,A -85,B 0,C 180,E1 -1024.327,E2 -1024.327} C_VEL
LIN {X 0,Y 746.379,Z 564.437,A -85,B 0,C 180,E1 -1026.914,E2 -1026.914} C_VEL
LIN {X 0,Y 746.372,Z 564.438,A -85,B 0,C 180,E1 -1028.96,E2 -1028.96} C_VEL
LIN {X 0,Y 746.39,Z 564.438,A -85,B 0,C 180,E1 -1031.345,E2 -1031.345} C_VEL
LIN {X 0,Y 746.363,Z 564.452,A -85,B 0,C 180,E1 -1033.985,E2 -1033.985} C_VEL
LIN {X 0,Y 746.367,Z 564.445,A -85,B 0,C 180,E1 -1036.271,E2 -1036.271} C_VEL
LIN {X 0,Y 746.392,Z 564.436,A -85,B 0,C 180,E1 -1038.936,E2 -1038.936} C_VEL
LIN {X 0,Y 746.368,Z 564.439,A -85,B 0,C 180,E1 -1041.163,E2 -1041.163} C_VEL
LIN {X 0,Y 746.352,Z 564.45,A -85,B 0,C 180,E1 -1043.755,E2 -1043.755} C_VEL
LIN {X 0,Y 746.366,Z 564.448,A -85,B 0,C 180,E1 -1045.731,E2 -1045.731} C_VEL
LIN {X 0,Y 746.371,Z 564.444,A -85,B 0,C 180,E1 -1048.296,E2 -1048.296} C_VEL
LIN {X 0,Y 746.365,Z 564.439,A -85,B 0,C 180,E1 -1050.791,E2 -1050.791} C_VEL
LIN {X 0,Y 746.354,Z 564.442,A -85,B 0,C 180,E1 -1053.226,E2 -1053.226} C_VEL
LIN {X 0,Y 746.341,Z 564.442,A -85,B 0,C 180,E1 -1055.019,E2 -1055.019} C_VEL
LIN {X 0,Y 746.336,Z 564.445,A -85,B 0,C 180,E1 -1057.37,E2 -1057.37} C_VEL
LIN {X 0,Y 746.387,Z 564.447,A -85,B 0,C 180,E1 -1059.792,E2 -1059.792} C_VEL
LIN {X 0,Y 746.374,Z 564.44,A -85,B 0,C 180,E1 -1062.524,E2 -1062.524} C_VEL
LIN {X 0,Y 746.356,Z 564.441,A -85,B 0,C 180,E1 -1065.159,E2 -1065.159} C_VEL
LIN {X 0,Y 746.364,Z 564.444,A -85,B 0,C 180,E1 -1067.535,E2 -1067.535} C_VEL
LIN {X 0,Y 746.401,Z 564.443,A -85,B 0,C 180,E1 -1070.18,E2 -1070.18} C_VEL
LIN {X 0,Y 746.402,Z 564.438,A -85,B 0,C 180,E1 -1072.451,E2 -1072.451} C_VEL
LIN {X 0,Y 746.355,Z 564.442,A -85,B 0,C 180,E1 -1074.615,E2 -1074.615} C_VEL
LIN {X 0,Y 746.335,Z 564.443,A -85,B 0,C 180,E1 -1076.772,E2 -1076.772} C_VEL
LIN {X 0,Y 746.357,Z 564.44,A -85,B 0,C 180,E1 -1078.925,E2 -1078.925} C_VEL
LIN {X 0,Y 746.351,Z 564.441,A -85,B 0,C 180,E1 -1081.076,E2 -1081.076} C_VEL
LIN {X 0,Y 746.362,Z 564.44,A -85,B 0,C 180,E1 -1082.69,E2 -1082.69} C_VEL
LIN {X 0,Y 746.382,Z 564.437,A -85,B 0,C 180,E1 -1084.845,E2 -1084.845} C_VEL
LIN {X 0,Y 746.357,Z 564.44,A -85,B 0,C 180,E1 -1087.008,E2 -1087.008} C_VEL
LIN {X 0,Y 746.351,Z 564.442,A -85,B 0,C 180,E1 -1089.181,E2 -1089.181} C_VEL
LIN {X 0,Y 746.339,Z 564.445,A -85,B 0,C 180,E1 -1091.367,E2 -1091.367} C_VEL
LIN {X 0,Y 746.346,Z 564.447,A -85,B 0,C 180,E1 -1093.57,E2 -1093.57} C_VEL
LIN {X 0,Y 746.353,Z 564.451,A -85,B 0,C 180,E1 -1095.793,E2 -1095.793} C_VEL
LIN {X 0,Y 746.349,Z 564.452,A -85,B 0,C 180,E1 -1098.041,E2 -1098.041} C_VEL
LIN {X 0,Y 746.371,Z 564.444,A -85,B 0,C 180,E1 -1100.318,E2 -1100.318} C_VEL
LIN {X 0,Y 746.346,Z 564.443,A -85,B 0,C 180,E1 -1102.63,E2 -1102.63} C_VEL
LIN {X 0,Y 746.314,Z 564.445,A -85,B 0,C 180,E1 -1104.983,E2 -1104.983} C_VEL
LIN {X 0,Y 746.342,Z 564.445,A -85,B 0,C 180,E1 -1107.379,E2 -1107.379} C_VEL
LIN {X 0,Y 746.37,Z 564.45,A -85,B 0,C 180,E1 -1109.827,E2 -1109.827} C_VEL
LIN {X 0,Y 746.358,Z 564.445,A -85,B 0,C 180,E1 -1112.367,E2 -1112.367} C_VEL
LIN {X 0,Y 746.327,Z 564.444,A -85,B 0,C 180,E1 -1114.925,E2 -1114.925} C_VEL
LIN {X 0,Y 746.337,Z 564.443,A -85,B 0,C 180,E1 -1117.086,E2 -1117.086} C_VEL
LIN {X 0,Y 746.343,Z 564.442,A -85,B 0,C 180,E1 -1118.961,E2 -1118.961} C_VEL
LIN {X 0,Y 746.367,Z 564.441,A -85,B 0,C 180,E1 -1121.342,E2 -1121.342} C_VEL
LIN {X 0,Y 746.349,Z 564.454,A -85,B 0,C 180,E1 -1123.986,E2 -1123.986} C_VEL
LIN {X 0,Y 746.347,Z 564.448,A -85,B 0,C 180,E1 -1126.273,E2 -1126.273} C_VEL
LIN {X 0,Y 746.339,Z 564.442,A -85,B 0,C 180,E1 -1128.932,E2 -1128.932} C_VEL
LIN {X 0,Y 746.341,Z 564.443,A -85,B 0,C 180,E1 -1131.165,E2 -1131.165} C_VEL
LIN {X 0,Y 746.347,Z 564.452,A -85,B 0,C 180,E1 -1133.814,E2 -1133.814} C_VEL
LIN {X 0,Y 746.335,Z 564.447,A -85,B 0,C 180,E1 -1136.377,E2 -1136.377} C_VEL
LIN {X 0,Y 746.329,Z 564.445,A -85,B 0,C 180,E1 -1138.655,E2 -1138.655} C_VEL
LIN {X 0,Y 746.325,Z 564.444,A -85,B 0,C 180,E1 -1140.789,E2 -1140.789} C_VEL
LIN {X 0,Y 746.34,Z 564.442,A -85,B 0,C 180,E1 -1143.072,E2 -1143.072} C_VEL
LIN {X 0,Y 746.304,Z 564.447,A -85,B 0,C 180,E1 -1145.017,E2 -1145.017} C_VEL
LIN {X 0,Y 746.309,Z 564.45,A -85,B 0,C 180,E1 -1147.369,E2 -1147.369} C_VEL
LIN {X 0,Y 746.33,Z 564.458,A -85,B 0,C 180,E1 -1149.142,E2 -1149.142} C_VEL
LIN {X 0,Y 746.592,Z 572.383,A -85,B 0,C 180,E1 -1150.132,E2 -1150.132} C_VEL
LIN {X 0,Y 746.548,Z 591.933,A -85,B 0,C 180,E1 -1152.528,E2 -1152.528} C_VEL
LIN {X 0,Y 746.409,Z 612.421,A -85,B 0,C 180,E1 -1155.005,E2 -1155.005} C_VEL
LIN {X 0,Y 746.388,Z 632.582,A -85,B 0,C 180,E1 -1157.416,E2 -1157.416} C_VEL
LIN {X 0,Y 746.32,Z 649.485,A -85,B 0,C 180,E1 -1159.421,E2 -1159.421} C_VEL
LIN {X 0,Y 746.54,Z 663.588,A -85,B 0,C 180,E1 -1159.56,E2 -1159.56} C_VEL
LIN {X 0,Y 746.474,Z 754.938,A -85,B 0,C 180,E1 -1160.447,E2 -1160.447} C_VEL
LIN {X 0,Y 746.461,Z 764.941,A -85,B 0,C 180,E1 -1160.6,E2 -1160.6} C_VEL
LIN {X 0,Y 746.435,Z 776.187,A -85,B 0,C 180,E1 -1160.855,E2 -1160.855} C_VEL
LIN {X 0,Y 746.463,Z 786.284,A -85,B 0,C 180,E1 -1161.161,E2 -1161.161} C_VEL
LIN {X 0,Y 746.426,Z 796.781,A -85,B 0,C 180,E1 -1161.569,E2 -1161.569} C_VEL
LIN {X 0,Y 746.401,Z 806.628,A -85,B 0,C 180,E1 -1162.044,E2 -1162.044} C_VEL
LIN {X 0,Y 746.364,Z 815.848,A -85,B 0,C 180,E1 -1162.586,E2 -1162.586} C_VEL
LIN {X 0,Y 746.335,Z 823.586,A -85,B 0,C 180,E1 -1163.128,E2 -1163.128} C_VEL
LIN {X 0,Y 746.297,Z 831.632,A -85,B 0,C 180,E1 -1163.804,E2 -1163.804} C_VEL
LIN {X 0,Y 746.276,Z 837.605,A -85,B 0,C 180,E1 -1164.395,E2 -1164.395} C_VEL
LIN {X 0,Y 746.283,Z 843.952,A -85,B 0,C 180,E1 -1165.154,E2 -1165.154} C_VEL
LIN {X 0,Y 746.294,Z 849.402,A -85,B 0,C 180,E1 -1165.964,E2 -1165.964} C_VEL
LIN {X 0,Y 746.252,Z 853.689,A -85,B 0,C 180,E1 -1166.772,E2 -1166.772} C_VEL
LIN {X 0,Y 746.246,Z 855.972,A -85,B 0,C 180,E1 -1167.31,E2 -1167.31} C_VEL
LIN {X 0,Y 746.232,Z 859.202,A -85,B 0,C 180,E1 -1168.386,E2 -1168.386} C_VEL
LIN {X 0,Y 746.238,Z 860.715,A -85,B 0,C 180,E1 -1169.462,E2 -1169.462} C_VEL
LIN {X 0,Y 746.236,Z 861,A -85,B 0,C 180,E1 -1170,E2 -1170} C_VEL
LIN {X 0,Y 746.241,Z 860.142,A -85,B 0,C 180,E1 -1171.076,E2 -1171.076} C_VEL
LIN {X 0,Y 746.232,Z 859.202,A -85,B 0,C 180,E1 -1171.614,E2 -1171.614} C_VEL
LIN {X 0,Y 746.246,Z 855.972,A -85,B 0,C 180,E1 -1172.69,E2 -1172.69} C_VEL
LIN {X 0,Y 746.24,Z 852.422,A -85,B 0,C 180,E1 -1173.498,E2 -1173.498} C_VEL
LIN {X 0,Y 746.245,Z 847.766,A -85,B 0,C 180,E1 -1174.307,E2 -1174.307} C_VEL
LIN {X 0,Y 746.302,Z 841.854,A -85,B 0,C 180,E1 -1175.116,E2 -1175.116} C_VEL
LIN {X 0,Y 746.308,Z 834.464,A -85,B 0,C 180,E1 -1175.926,E2 -1175.926} C_VEL
LIN {X 0,Y 746.327,Z 826.97,A -85,B 0,C 180,E1 -1176.602,E2 -1176.602} C_VEL
LIN {X 0,Y 746.362,Z 819.886,A -85,B 0,C 180,E1 -1177.143,E2 -1177.143} C_VEL
LIN {X 0,Y 746.362,Z 811.478,A -85,B 0,C 180,E1 -1177.685,E2 -1177.685} C_VEL
LIN {X 0,Y 746.411,Z 801.222,A -85,B 0,C 180,E1 -1178.228,E2 -1178.228} C_VEL
LIN {X 0,Y 746.413,Z 791.826,A -85,B 0,C 180,E1 -1178.636,E2 -1178.636} C_VEL
LIN {X 0,Y 746.445,Z 780.974,A -85,B 0,C 180,E1 -1179.009,E2 -1179.009} C_VEL
LIN {X 0,Y 746.431,Z 769.892,A -85,B 0,C 180,E1 -1179.299,E2 -1179.299} C_VEL
LIN {X 0,Y 746.465,Z 758.808,A -85,B 0,C 180,E1 -1179.503,E2 -1179.503} C_VEL
LIN {X 0,Y 746.474,Z 740.446,A -85,B 0,C 180,E1 -1179.705,E2 -1179.705} C_VEL
LIN {X 0,Y 746.388,Z 650.196,A -85,B 0,C 180,E1 -1180.57,E2 -1180.57} C_VEL
LIN {X 0,Y 746.32,Z 649.483,A -85,B 0,C 180,E1 -1180.58,E2 -1180.58} C_VEL
LIN {X 0,Y 746.41,Z 630.195,A -85,B 0,C 180,E1 -1182.867,E2 -1182.867} C_VEL
LIN {X 0,Y 746.422,Z 610.44,A -85,B 0,C 180,E1 -1185.234,E2 -1185.234} C_VEL
LIN {X 0,Y 746.525,Z 590.774,A -85,B 0,C 180,E1 -1187.614,E2 -1187.614} C_VEL
LIN {X 0,Y 746.608,Z 571.335,A -85,B 0,C 180,E1 -1189.997,E2 -1189.997} C_VEL
LIN {X 0,Y 746.33,Z 564.456,A -85,B 0,C 180,E1 -1190.858,E2 -1190.858} C_VEL
LIN {X 0,Y 746.301,Z 564.45,A -85,B 0,C 180,E1 -1193.216,E2 -1193.216} C_VEL
LIN {X 0,Y 746.362,Z 564.45,A -85,B 0,C 180,E1 -1195.719,E2 -1195.719} C_VEL
LIN {X 0,Y 746.373,Z 564.447,A -85,B 0,C 180,E1 -1198.097,E2 -1198.097} C_VEL
LIN {X 0,Y 746.344,Z 564.444,A -85,B 0,C 180,E1 -1200.45,E2 -1200.45} C_VEL
LIN {X 0,Y 746.35,Z 564.443,A -85,B 0,C 180,E1 -1202.979,E2 -1202.979} C_VEL
LIN {X 0,Y 746.366,Z 564.453,A -85,B 0,C 180,E1 -1205.581,E2 -1205.581} C_VEL
LIN {X 0,Y 746.357,Z 564.441,A -85,B 0,C 180,E1 -1208.273,E2 -1208.273} C_VEL
LIN {X 0,Y 746.338,Z 564.443,A -85,B 0,C 180,E1 -1210.519,E2 -1210.519} C_VEL
LIN {X 0,Y 746.34,Z 564.443,A -85,B 0,C 180,E1 -1212.511,E2 -1212.511} C_VEL
LIN {X 0,Y 746.356,Z 564.444,A -85,B 0,C 180,E1 -1214.738,E2 -1214.738} C_VEL
LIN {X 0,Y 746.363,Z 564.45,A -85,B 0,C 180,E1 -1217.056,E2 -1217.056} C_VEL
LIN {X 0,Y 746.389,Z 564.443,A -85,B 0,C 180,E1 -1219.477,E2 -1219.477} C_VEL
LIN {X 0,Y 746.363,Z 564.44,A -85,B 0,C 180,E1 -1222.029,E2 -1222.029} C_VEL
LIN {X 0,Y 746.375,Z 564.441,A -85,B 0,C 180,E1 -1224.42,E2 -1224.42} C_VEL
LIN {X 0,Y 746.375,Z 564.449,A -85,B 0,C 180,E1 -1227.023,E2 -1227.023} C_VEL
LIN {X 0,Y 746.368,Z 564.441,A -85,B 0,C 180,E1 -1229.551,E2 -1229.551} C_VEL
LIN {X 0,Y 746.392,Z 564.438,A -85,B 0,C 180,E1 -1232.016,E2 -1232.016} C_VEL
LIN {X 0,Y 746.402,Z 564.443,A -85,B 0,C 180,E1 -1234.426,E2 -1234.426} C_VEL
LIN {X 0,Y 746.364,Z 564.448,A -85,B 0,C 180,E1 -1236.884,E2 -1236.884} C_VEL
LIN {X 0,Y 746.369,Z 564.442,A -85,B 0,C 180,E1 -1239.107,E2 -1239.107} C_VEL
LIN {X 0,Y 746.377,Z 564.439,A -85,B 0,C 180,E1 -1241.414,E2 -1241.414} C_VEL
LIN {X 0,Y 746.372,Z 564.44,A -85,B 0,C 180,E1 -1243.648,E2 -1243.648} C_VEL
LIN {X 0,Y 746.356,Z 564.446,A -85,B 0,C 180,E1 -1245.877,E2 -1245.877} C_VEL
LIN {X 0,Y 746.384,Z 564.447,A -85,B 0,C 180,E1 -1248.085,E2 -1248.085} C_VEL
LIN {X 0,Y 746.373,Z 564.452,A -85,B 0,C 180,E1 -1250.275,E2 -1250.275} C_VEL
LIN {X 0,Y 746.397,Z 564.494,A -85,B 0,C 180,E1 -1251.534,E2 -1251.534} C_VEL
LIN {X 0,Y 746.439,Z 580.313,A -85,B 0,C 180,E1 -1253.805,E2 -1253.805} C_VEL
LIN {X 0,Y 746.364,Z 597.451,A -85,B 0,C 180,E1 -1256.233,E2 -1256.233} C_VEL
LIN {X 0,Y 746.33,Z 614.717,A -85,B 0,C 180,E1 -1258.655,E2 -1258.655} C_VEL
LIN {X 0,Y 746.327,Z 620.707,A -85,B 0,C 180,E1 -1259.479,E2 -1259.479} C_VEL
LIN {X 0,Y 746.588,Z 632.605,A -85,B 0,C 180,E1 -1259.597,E2 -1259.597} C_VEL
LIN {X 0,Y 746.459,Z 726.007,A -85,B 0,C 180,E1 -1260.504,E2 -1260.504} C_VEL
LIN {X 0,Y 746.439,Z 736.355,A -85,B 0,C 180,E1 -1260.672,E2 -1260.672} C_VEL
LIN {X 0,Y 746.433,Z 746.495,A -85,B 0,C 180,E1 -1260.907,E2 -1260.907} C_VEL
LIN {X 0,Y 746.453,Z 756.423,A -85,B 0,C 180,E1 -1261.21,E2 -1261.21} C_VEL
LIN {X 0,Y 746.424,Z 766.792,A -85,B 0,C 180,E1 -1261.613,E2 -1261.613} C_VEL
LIN {X 0,Y 746.369,Z 776.576,A -85,B 0,C 180,E1 -1262.084,E2 -1262.084} C_VEL
LIN {X 0,Y 746.346,Z 785.738,A -85,B 0,C 180,E1 -1262.622,E2 -1262.622} C_VEL
LIN {X 0,Y 746.316,Z 794.308,A -85,B 0,C 180,E1 -1263.228,E2 -1263.228} C_VEL
LIN {X 0,Y 746.292,Z 800.787,A -85,B 0,C 180,E1 -1263.767,E2 -1263.767} C_VEL
LIN {X 0,Y 746.276,Z 807.635,A -85,B 0,C 180,E1 -1264.441,E2 -1264.441} C_VEL
LIN {X 0,Y 746.3,Z 813.361,A -85,B 0,C 180,E1 -1265.115,E2 -1265.115} C_VEL
LIN {X 0,Y 746.268,Z 818.956,A -85,B 0,C 180,E1 -1265.926,E2 -1265.926} C_VEL
LIN {X 0,Y 746.26,Z 823.36,A -85,B 0,C 180,E1 -1266.738,E2 -1266.738} C_VEL
LIN {X 0,Y 746.253,Z 826.715,A -85,B 0,C 180,E1 -1267.551,E2 -1267.551} C_VEL
LIN {X 0,Y 746.241,Z 829.578,A -85,B 0,C 180,E1 -1268.637,E2 -1268.637} C_VEL
LIN {X 0,Y 746.256,Z 830.485,A -85,B 0,C 180,E1 -1269.181,E2 -1269.181} C_VEL
LIN {X 0,Y 746.222,Z 830.876,A -85,B 0,C 180,E1 -1270.327,E2 -1270.327} C_VEL
LIN {X 0,Y 746.223,Z 830.584,A -85,B 0,C 180,E1 -1270.82,E2 -1270.82} C_VEL
LIN {X 0,Y 746.24,Z 828.569,A -85,B 0,C 180,E1 -1271.917,E2 -1271.917} C_VEL
LIN {X 0,Y 746.236,Z 826.264,A -85,B 0,C 180,E1 -1272.65,E2 -1272.65} C_VEL
LIN {X 0,Y 745.566,Z 824.557,A -85,B 0,C 180,E1 -1273.079,E2 -1273.079} C_VEL
LIN {X 0,Y 743.965,Z 822.74,A -85,B 0,C 180,E1 -1273.494,E2 -1273.494} C_VEL
LIN {X 0,Y 739.8,Z 817.451,A -85,B 0,C 180,E1 -1274.437,E2 -1274.437} C_VEL
LIN {X 0,Y 739.189,Z 814.634,A -85,B 0,C 180,E1 -1274.843,E2 -1274.843} C_VEL
LIN {X 0,Y 739.229,Z 807.954,A -85,B 0,C 180,E1 -1275.667,E2 -1275.667} C_VEL
LIN {X 0,Y 739.257,Z 799.374,A -85,B 0,C 180,E1 -1276.514,E2 -1276.514} C_VEL
LIN {X 0,Y 739.302,Z 789.382,A -85,B 0,C 180,E1 -1277.293,E2 -1277.293} C_VEL
LIN {X 0,Y 739.348,Z 780.508,A -85,B 0,C 180,E1 -1277.861,E2 -1277.861} C_VEL
LIN {X 0,Y 739.388,Z 771.516,A -85,B 0,C 180,E1 -1278.34,E2 -1278.34} C_VEL
LIN {X 0,Y 739.418,Z 761.201,A -85,B 0,C 180,E1 -1278.788,E2 -1278.788} C_VEL
LIN {X 0,Y 739.44,Z 750.827,A -85,B 0,C 180,E1 -1279.147,E2 -1279.147} C_VEL
LIN {X 0,Y 739.46,Z 739.945,A -85,B 0,C 180,E1 -1279.433,E2 -1279.433} C_VEL
LIN {X 0,Y 739.528,Z 728.223,A -85,B 0,C 180,E1 -1279.648,E2 -1279.648} C_VEL
LIN {X 0,Y 739.539,Z 706.327,A -85,B 0,C 180,E1 -1279.882,E2 -1279.882} C_VEL
LIN {X 0,Y 739.43,Z 621.997,A -85,B 0,C 180,E1 -1280.698,E2 -1280.698} C_VEL
LIN {X 0,Y 739.251,Z 620.562,A -85,B 0,C 180,E1 -1280.722,E2 -1280.722} C_VEL
LIN {X 0,Y 739.314,Z 604.151,A -85,B 0,C 180,E1 -1283.039,E2 -1283.039} C_VEL
LIN {X 0,Y 739.361,Z 586.651,A -85,B 0,C 180,E1 -1285.534,E2 -1285.534} C_VEL
LIN {X 0,Y 739.453,Z 569.893,A -85,B 0,C 180,E1 -1287.95,E2 -1287.95} C_VEL
LIN {X 0,Y 739.33,Z 565.321,A -85,B 0,C 180,E1 -1288.622,E2 -1288.622} C_VEL
LIN {X 0,Y 739.309,Z 565.319,A -85,B 0,C 180,E1 -1290.771,E2 -1290.771} C_VEL
LIN {X 0,Y 739.351,Z 565.317,A -85,B 0,C 180,E1 -1293.52,E2 -1293.52} C_VEL
LIN {X 0,Y 739.316,Z 565.331,A -85,B 0,C 180,E1 -1295.972,E2 -1295.972} C_VEL
LIN {X 0,Y 739.335,Z 565.324,A -85,B 0,C 180,E1 -1298.155,E2 -1298.155} C_VEL
LIN {X 0,Y 739.335,Z 565.316,A -85,B 0,C 180,E1 -1300.719,E2 -1300.719} C_VEL
LIN {X 0,Y 739.327,Z 565.316,A -85,B 0,C 180,E1 -1303.155,E2 -1303.155} C_VEL
LIN {X 0,Y 739.338,Z 565.318,A -85,B 0,C 180,E1 -1305.487,E2 -1305.487} C_VEL
LIN {X 0,Y 739.308,Z 565.327,A -85,B 0,C 180,E1 -1307.726,E2 -1307.726} C_VEL
LIN {X 0,Y 739.323,Z 565.326,A -85,B 0,C 180,E1 -1310.121,E2 -1310.121} C_VEL
LIN {X 0,Y 739.315,Z 565.33,A -85,B 0,C 180,E1 -1311.988,E2 -1311.988} C_VEL
LIN {X 0,Y 739.321,Z 565.317,A -85,B 0,C 180,E1 -1314.695,E2 -1314.695} C_VEL
LIN {X 0,Y 739.333,Z 565.317,A -85,B 0,C 180,E1 -1317.315,E2 -1317.315} C_VEL
LIN {X 0,Y 739.319,Z 565.328,A -85,B 0,C 180,E1 -1319.859,E2 -1319.859} C_VEL
LIN {X 0,Y 739.321,Z 565.322,A -85,B 0,C 180,E1 -1322.339,E2 -1322.339} C_VEL
LIN {X 0,Y 739.324,Z 565.317,A -85,B 0,C 180,E1 -1324.765,E2 -1324.765} C_VEL
LIN {X 0,Y 739.318,Z 565.317,A -85,B 0,C 180,E1 -1327.142,E2 -1327.142} C_VEL
LIN {X 0,Y 739.33,Z 565.323,A -85,B 0,C 180,E1 -1329.705,E2 -1329.705} C_VEL
LIN {X 0,Y 739.324,Z 565.326,A -85,B 0,C 180,E1 -1331.781,E2 -1331.781} C_VEL
LIN {X 0,Y 739.338,Z 565.326,A -85,B 0,C 180,E1 -1334.053,E2 -1334.053} C_VEL
LIN {X 0,Y 739.309,Z 565.324,A -85,B 0,C 180,E1 -1336.299,E2 -1336.299} C_VEL
LIN {X 0,Y 739.333,Z 565.318,A -85,B 0,C 180,E1 -1338.524,E2 -1338.524} C_VEL
LIN {X 0,Y 739.348,Z 565.314,A -85,B 0,C 180,E1 -1340.732,E2 -1340.732} C_VEL
LIN {X 0,Y 739.367,Z 565.311,A -85,B 0,C 180,E1 -1342.926,E2 -1342.926} C_VEL
LIN {X 0,Y 739.391,Z 565.315,A -85,B 0,C 180,E1 -1345.653,E2 -1345.653} C_VEL
LIN {X 0,Y 739.361,Z 565.316,A -85,B 0,C 180,E1 -1348.371,E2 -1348.371} C_VEL
LIN {X 0,Y 739.336,Z 565.317,A -85,B 0,C 180,E1 -1350.543,E2 -1350.543} C_VEL
LIN {X 0,Y 739.317,Z 565.318,A -85,B 0,C 180,E1 -1352.715,E2 -1352.715} C_VEL
LIN {X 0,Y 739.374,Z 565.31,A -85,B 0,C 180,E1 -1354.891,E2 -1354.891} C_VEL
LIN {X 0,Y 739.331,Z 565.322,A -85,B 0,C 180,E1 -1357.622,E2 -1357.622} C_VEL
LIN {X 0,Y 739.346,Z 565.325,A -85,B 0,C 180,E1 -1359.846,E2 -1359.846} C_VEL
LIN {X 0,Y 739.337,Z 565.326,A -85,B 0,C 180,E1 -1362.03,E2 -1362.03} C_VEL
LIN {X 0,Y 739.362,Z 565.311,A -85,B 0,C 180,E1 -1364.917,E2 -1364.917} C_VEL
LIN {X 0,Y 739.355,Z 565.313,A -85,B 0,C 180,E1 -1367.079,E2 -1367.079} C_VEL
LIN {X 0,Y 739.327,Z 565.318,A -85,B 0,C 180,E1 -1369.365,E2 -1369.365} C_VEL
LIN {X 0,Y 739.333,Z 565.325,A -85,B 0,C 180,E1 -1371.807,E2 -1371.807} C_VEL
LIN {X 0,Y 739.31,Z 565.329,A -85,B 0,C 180,E1 -1374.041,E2 -1374.041} C_VEL
LIN {X 0,Y 739.318,Z 565.321,A -85,B 0,C 180,E1 -1376.442,E2 -1376.442} C_VEL
LIN {X 0,Y 739.342,Z 565.314,A -85,B 0,C 180,E1 -1378.892,E2 -1378.892} C_VEL
LIN {X 0,Y 739.318,Z 565.32,A -85,B 0,C 180,E1 -1381.405,E2 -1381.405} C_VEL
LIN {X 0,Y 739.349,Z 565.318,A -85,B 0,C 180,E1 -1383.521,E2 -1383.521} C_VEL
LIN {X 0,Y 739.316,Z 565.331,A -85,B 0,C 180,E1 -1385.973,E2 -1385.973} C_VEL
LIN {X 0,Y 739.338,Z 565.323,A -85,B 0,C 180,E1 -1388.156,E2 -1388.156} C_VEL
LIN {X 0,Y 739.342,Z 565.314,A -85,B 0,C 180,E1 -1390.821,E2 -1390.821} C_VEL
LIN {X 0,Y 739.325,Z 565.317,A -85,B 0,C 180,E1 -1393.156,E2 -1393.156} C_VEL
LIN {X 0,Y 739.328,Z 565.32,A -85,B 0,C 180,E1 -1395.487,E2 -1395.487} C_VEL
LIN {X 0,Y 739.301,Z 565.328,A -85,B 0,C 180,E1 -1397.726,E2 -1397.726} C_VEL
LIN {X 0,Y 739.321,Z 565.326,A -85,B 0,C 180,E1 -1400.122,E2 -1400.122} C_VEL
LIN {X 0,Y 739.323,Z 565.317,A -85,B 0,C 180,E1 -1402.675,E2 -1402.675} C_VEL
LIN {X 0,Y 739.335,Z 565.317,A -85,B 0,C 180,E1 -1405.359,E2 -1405.359} C_VEL
LIN {X 0,Y 739.321,Z 565.321,A -85,B 0,C 180,E1 -1407.48,E2 -1407.48} C_VEL
LIN {X 0,Y 739.311,Z 565.33,A -85,B 0,C 180,E1 -1409.859,E2 -1409.859} C_VEL
LIN {X 0,Y 739.315,Z 565.322,A -85,B 0,C 180,E1 -1412.34,E2 -1412.34} C_VEL
LIN {X 0,Y 739.327,Z 565.316,A -85,B 0,C 180,E1 -1414.765,E2 -1414.765} C_VEL
LIN {X 0,Y 739.3,Z 565.32,A -85,B 0,C 180,E1 -1417.142,E2 -1417.142} C_VEL
LIN {X 0,Y 739.327,Z 565.32,A -85,B 0,C 180,E1 -1419.48,E2 -1419.48} C_VEL
LIN {X 0,Y 739.315,Z 565.327,A -85,B 0,C 180,E1 -1421.781,E2 -1421.781} C_VEL
LIN {X 0,Y 739.336,Z 565.326,A -85,B 0,C 180,E1 -1424.053,E2 -1424.053} C_VEL
LIN {X 0,Y 739.319,Z 565.323,A -85,B 0,C 180,E1 -1426.299,E2 -1426.299} C_VEL
LIN {X 0,Y 739.329,Z 565.318,A -85,B 0,C 180,E1 -1428.524,E2 -1428.524} C_VEL
LIN {X 0,Y 739.34,Z 565.315,A -85,B 0,C 180,E1 -1430.732,E2 -1430.732} C_VEL
LIN {X 0,Y 739.319,Z 565.317,A -85,B 0,C 180,E1 -1432.925,E2 -1432.925} C_VEL
LIN {X 0,Y 739.336,Z 565.315,A -85,B 0,C 180,E1 -1435.109,E2 -1435.109} C_VEL
LIN {X 0,Y 739.362,Z 565.323,A -85,B 0,C 180,E1 -1437.828,E2 -1437.828} C_VEL
LIN {X 0,Y 739.346,Z 565.316,A -85,B 0,C 180,E1 -1440.543,E2 -1440.543} C_VEL
LIN {X 0,Y 739.313,Z 565.318,A -85,B 0,C 180,E1 -1442.715,E2 -1442.715} C_VEL
LIN {X 0,Y 739.352,Z 565.313,A -85,B 0,C 180,E1 -1444.891,E2 -1444.891} C_VEL
LIN {X 0,Y 739.31,Z 565.318,A -85,B 0,C 180,E1 -1447.075,E2 -1447.075} C_VEL
LIN {X 0,Y 739.324,Z 565.318,A -85,B 0,C 180,E1 -1449.269,E2 -1449.269} C_VEL
LIN {X 0,Y 739.296,Z 565.324,A -85,B 0,C 180,E1 -1451.476,E2 -1451.476} C_VEL
LIN {X 0,Y 739.303,Z 565.319,A -85,B 0,C 180,E1 -1453.143,E2 -1453.143} C_VEL
LIN {X 0,Y 739.302,Z 565.322,A -85,B 0,C 180,E1 -1455.384,E2 -1455.384} C_VEL
LIN {X 0,Y 739.318,Z 565.324,A -85,B 0,C 180,E1 -1457.648,E2 -1457.648} C_VEL
LIN {X 0,Y 739.333,Z 565.321,A -85,B 0,C 180,E1 -1460.294,E2 -1460.294} C_VEL
LIN {X 0,Y 739.295,Z 565.32,A -85,B 0,C 180,E1 -1462.858,E2 -1462.858} C_VEL
LIN {X 0,Y 739.295,Z 565.321,A -85,B 0,C 180,E1 -1465.236,E2 -1465.236} C_VEL
LIN {X 0,Y 739.308,Z 565.326,A -85,B 0,C 180,E1 -1467.661,E2 -1467.661} C_VEL
LIN {X 0,Y 739.313,Z 565.326,A -85,B 0,C 180,E1 -1470.141,E2 -1470.141} C_VEL
LIN {X 0,Y 739.291,Z 565.321,A -85,B 0,C 180,E1 -1472.687,E2 -1472.687} C_VEL
LIN {X 0,Y 739.305,Z 565.32,A -85,B 0,C 180,E1 -1474.643,E2 -1474.643} C_VEL
LIN {X 0,Y 739.31,Z 565.32,A -85,B 0,C 180,E1 -1477.326,E2 -1477.326} C_VEL
LIN {X 0,Y 739.288,Z 565.324,A -85,B 0,C 180,E1 -1479.405,E2 -1479.405} C_VEL
LIN {X 0,Y 739.325,Z 565.321,A -85,B 0,C 180,E1 -1481.543,E2 -1481.543} C_VEL
LIN {X 0,Y 739.321,Z 565.33,A -85,B 0,C 180,E1 -1483.943,E2 -1483.943} C_VEL
LIN {X 0,Y 739.301,Z 565.326,A -85,B 0,C 180,E1 -1486.241,E2 -1486.241} C_VEL
LIN {X 0,Y 739.324,Z 565.319,A -85,B 0,C 180,E1 -1488.457,E2 -1488.457} C_VEL
LIN {X 0,Y 739.317,Z 565.317,A -85,B 0,C 180,E1 -1490.976,E2 -1490.976} C_VEL
LIN {X 0,Y 739.284,Z 565.328,A -85,B 0,C 180,E1 -1493.643,E2 -1493.643} C_VEL
LIN {X 0,Y 739.321,Z 565.319,A -85,B 0,C 180,E1 -1496.483,E2 -1496.483} C_VEL
LIN {X 0,Y 739.294,Z 565.322,A -85,B 0,C 180,E1 -1498.594,E2 -1498.594} C_VEL
LIN {X 0,Y 739.304,Z 565.32,A -85,B 0,C 180,E1 -1500.65,E2 -1500.65} C_VEL
LIN {X 0,Y 739.29,Z 565.32,A -85,B 0,C 180,E1 -1502.949,E2 -1502.949} C_VEL
LIN {X 0,Y 739.308,Z 565.322,A -85,B 0,C 180,E1 -1505.441,E2 -1505.441} C_VEL
LIN {X 0,Y 739.317,Z 565.326,A -85,B 0,C 180,E1 -1508.316,E2 -1508.316} C_VEL
LIN {X 0,Y 739.323,Z 565.47,A -85,B 0,C 180,E1 -1509.062,E2 -1509.062} C_VEL
LIN {X 0,Y 739.651,Z 571.717,A -85,B 0,C 180,E1 -1509.854,E2 -1509.854} C_VEL
LIN {X 0,Y 739.538,Z 591.933,A -85,B 0,C 180,E1 -1512.357,E2 -1512.357} C_VEL
LIN {X 0,Y 739.388,Z 612.737,A -85,B 0,C 180,E1 -1514.897,E2 -1514.897} C_VEL
LIN {X 0,Y 739.351,Z 631.496,A -85,B 0,C 180,E1 -1517.164,E2 -1517.164} C_VEL
LIN {X 0,Y 739.273,Z 649.485,A -85,B 0,C 180,E1 -1519.319,E2 -1519.319} C_VEL
LIN {X 0,Y 739.571,Z 656.457,A -85,B 0,C 180,E1 -1519.392,E2 -1519.392} C_VEL
LIN {X 0,Y 739.481,Z 754.889,A -85,B 0,C 180,E1 -1520.355,E2 -1520.355} C_VEL
LIN {X 0,Y 739.467,Z 765.392,A -85,B 0,C 180,E1 -1520.519,E2 -1520.519} C_VEL
LIN {X 0,Y 739.435,Z 776.187,A -85,B 0,C 180,E1 -1520.767,E2 -1520.767} C_VEL
LIN {X 0,Y 739.449,Z 786.282,A -85,B 0,C 180,E1 -1521.077,E2 -1521.077} C_VEL
LIN {X 0,Y 739.391,Z 796.778,A -85,B 0,C 180,E1 -1521.488,E2 -1521.488} C_VEL
LIN {X 0,Y 739.348,Z 806.626,A -85,B 0,C 180,E1 -1521.967,E2 -1521.967} C_VEL
LIN {X 0,Y 739.3,Z 815.848,A -85,B 0,C 180,E1 -1522.515,E2 -1522.515} C_VEL
LIN {X 0,Y 739.274,Z 823.585,A -85,B 0,C 180,E1 -1523.062,E2 -1523.062} C_VEL
LIN {X 0,Y 739.23,Z 831.632,A -85,B 0,C 180,E1 -1523.744,E2 -1523.744} C_VEL
LIN {X 0,Y 739.188,Z 838.402,A -85,B 0,C 180,E1 -1524.434,E2 -1524.434} C_VEL
LIN {X 0,Y 739.213,Z 843.953,A -85,B 0,C 180,E1 -1525.108,E2 -1525.108} C_VEL
LIN {X 0,Y 739.218,Z 849.402,A -85,B 0,C 180,E1 -1525.925,E2 -1525.925} C_VEL
LIN {X 0,Y 739.16,Z 853.689,A -85,B 0,C 180,E1 -1526.741,E2 -1526.741} C_VEL
LIN {X 0,Y 739.167,Z 855.973,A -85,B 0,C 180,E1 -1527.284,E2 -1527.284} C_VEL
LIN {X 0,Y 739.131,Z 859.2,A -85,B 0,C 180,E1 -1528.371,E2 -1528.371} C_VEL
LIN {X 0,Y 739.139,Z 860.715,A -85,B 0,C 180,E1 -1529.457,E2 -1529.457} C_VEL
LIN {X 0,Y 739.137,Z 861,A -85,B 0,C 180,E1 -1530,E2 -1530} C_VEL
LIN {X 0,Y 739.141,Z 860.143,A -85,B 0,C 180,E1 -1531.086,E2 -1531.086} C_VEL
LIN {X 0,Y 739.132,Z 859.201,A -85,B 0,C 180,E1 -1531.629,E2 -1531.629} C_VEL
LIN {X 0,Y 739.167,Z 855.973,A -85,B 0,C 180,E1 -1532.716,E2 -1532.716} C_VEL
LIN {X 0,Y 739.157,Z 852.422,A -85,B 0,C 180,E1 -1533.532,E2 -1533.532} C_VEL
LIN {X 0,Y 739.152,Z 847.766,A -85,B 0,C 180,E1 -1534.348,E2 -1534.348} C_VEL
LIN {X 0,Y 739.231,Z 841.854,A -85,B 0,C 180,E1 -1535.165,E2 -1535.165} C_VEL
LIN {X 0,Y 739.237,Z 834.464,A -85,B 0,C 180,E1 -1535.983,E2 -1535.983} C_VEL
LIN {X 0,Y 739.278,Z 826.97,A -85,B 0,C 180,E1 -1536.665,E2 -1536.665} C_VEL
LIN {X 0,Y 739.326,Z 819.887,A -85,B 0,C 180,E1 -1537.212,E2 -1537.212} C_VEL
LIN {X 0,Y 739.318,Z 811.481,A -85,B 0,C 180,E1 -1537.759,E2 -1537.759} C_VEL
LIN {X 0,Y 739.365,Z 801.225,A -85,B 0,C 180,E1 -1538.307,E2 -1538.307} C_VEL
LIN {X 0,Y 739.401,Z 791.83,A -85,B 0,C 180,E1 -1538.718,E2 -1538.718} C_VEL
LIN {X 0,Y 739.434,Z 780.976,A -85,B 0,C 180,E1 -1539.095,E2 -1539.095} C_VEL
LIN {X 0,Y 739.43,Z 770.096,A -85,B 0,C 180,E1 -1539.383,E2 -1539.383} C_VEL
LIN {X 0,Y 739.488,Z 759.671,A -85,B 0,C 180,E1 -1539.582,E2 -1539.582} C_VEL
LIN {X 0,Y 739.503,Z 742.524,A -85,B 0,C 180,E1 -1539.777,E2 -1539.777} C_VEL
LIN {X 0,Y 739.412,Z 650.642,A -85,B 0,C 180,E1 -1540.667,E2 -1540.667} C_VEL
LIN {X 0,Y 739.273,Z 649.483,A -85,B 0,C 180,E1 -1540.682,E2 -1540.682} C_VEL
LIN {X 0,Y 739.348,Z 630.108,A -85,B 0,C 180,E1 -1543.003,E2 -1543.003} C_VEL
LIN {X 0,Y 739.409,Z 611.581,A -85,B 0,C 180,E1 -1545.243,E2 -1545.243} C_VEL
LIN {X 0,Y 739.538,Z 591.931,A -85,B 0,C 180,E1 -1547.643,E2 -1547.643} C_VEL
LIN {X 0,Y 739.652,Z 571.713,A -85,B 0,C 180,E1 -1550.146,E2 -1550.146} C_VEL
LIN {X 0,Y 739.324,Z 565.469,A -85,B 0,C 180,E1 -1550.938,E2 -1550.938} C_VEL
LIN {X 0,Y 739.268,Z 565.329,A -85,B 0,C 180,E1 -1553.45,E2 -1553.45} C_VEL
LIN {X 0,Y 739.325,Z 565.33,A -85,B 0,C 180,E1 -1555.837,E2 -1555.837} C_VEL
LIN {X 0,Y 739.307,Z 565.324,A -85,B 0,C 180,E1 -1558.276,E2 -1558.276} C_VEL
LIN {X 0,Y 739.292,Z 565.322,A -85,B 0,C 180,E1 -1560.772,E2 -1560.772} C_VEL
LIN {X 0,Y 739.344,Z 565.325,A -85,B 0,C 180,E1 -1563.52,E2 -1563.52} C_VEL
LIN {X 0,Y 739.3,Z 565.321,A -85,B 0,C 180,E1 -1566.358,E2 -1566.358} C_VEL
LIN {X 0,Y 739.337,Z 565.319,A -85,B 0,C 180,E1 -1569.026,E2 -1569.026} C_VEL
LIN {X 0,Y 739.352,Z 565.323,A -85,B 0,C 180,E1 -1571.546,E2 -1571.546} C_VEL
LIN {X 0,Y 739.329,Z 565.318,A -85,B 0,C 180,E1 -1573.943,E2 -1573.943} C_VEL
LIN {X 0,Y 739.314,Z 565.319,A -85,B 0,C 180,E1 -1576.242,E2 -1576.242} C_VEL
LIN {X 0,Y 739.356,Z 565.314,A -85,B 0,C 180,E1 -1578.459,E2 -1578.459} C_VEL
LIN {X 0,Y 739.348,Z 565.323,A -85,B 0,C 180,E1 -1581.298,E2 -1581.298} C_VEL
LIN {X 0,Y 739.32,Z 565.318,A -85,B 0,C 180,E1 -1584.027,E2 -1584.027} C_VEL
LIN {X 0,Y 739.354,Z 565.317,A -85,B 0,C 180,E1 -1586.48,E2 -1586.48} C_VEL
LIN {X 0,Y 739.326,Z 565.322,A -85,B 0,C 180,E1 -1589.229,E2 -1589.229} C_VEL
LIN {X 0,Y 739.353,Z 565.314,A -85,B 0,C 180,E1 -1591.771,E2 -1591.771} C_VEL
LIN {X 0,Y 739.364,Z 565.315,A -85,B 0,C 180,E1 -1594.165,E2 -1594.165} C_VEL
LIN {X 0,Y 739.317,Z 565.328,A -85,B 0,C 180,E1 -1596.781,E2 -1596.781} C_VEL
LIN {X 0,Y 739.341,Z 565.321,A -85,B 0,C 180,E1 -1598.899,E2 -1598.899} C_VEL
LIN {X 0,Y 739.352,Z 565.315,A -85,B 0,C 180,E1 -1601.33,E2 -1601.33} C_VEL
LIN {X 0,Y 739.339,Z 565.322,A -85,B 0,C 180,E1 -1604.053,E2 -1604.053} C_VEL
LIN {X 0,Y 739.308,Z 565.332,A -85,B 0,C 180,E1 -1606.299,E2 -1606.299} C_VEL
LIN {X 0,Y 739.304,Z 565.328,A -85,B 0,C 180,E1 -1608.524,E2 -1608.524} C_VEL
LIN {X 0,Y 739.326,Z 565.322,A -85,B 0,C 180,E1 -1610.731,E2 -1610.731} C_VEL
LIN {X 0,Y 739.351,Z 565.426,A -85,B 0,C 180,E1 -1611.487,E2 -1611.487} C_VEL
LIN {X 0,Y 739.432,Z 579.107,A -85,B 0,C 180,E1 -1613.473,E2 -1613.473} C_VEL
LIN {X 0,Y 739.362,Z 596.228,A -85,B 0,C 180,E1 -1615.925,E2 -1615.925} C_VEL
LIN {X 0,Y 739.293,Z 613.481,A -85,B 0,C 180,E1 -1618.371,E2 -1618.371} C_VEL
LIN {X 0,Y 739.286,Z 620.586,A -85,B 0,C 180,E1 -1619.372,E2 -1619.372} C_VEL
LIN {X 0,Y 739.633,Z 630.216,A -85,B 0,C 180,E1 -1619.474,E2 -1619.474} C_VEL
LIN {X 0,Y 739.458,Z 725.613,A -85,B 0,C 180,E1 -1620.407,E2 -1620.407} C_VEL
LIN {X 0,Y 739.43,Z 736.926,A -85,B 0,C 180,E1 -1620.593,E2 -1620.593} C_VEL
LIN {X 0,Y 739.419,Z 747.498,A -85,B 0,C 180,E1 -1620.848,E2 -1620.848} C_VEL
LIN {X 0,Y 739.439,Z 757.199,A -85,B 0,C 180,E1 -1621.153,E2 -1621.153} C_VEL
LIN {X 0,Y 739.386,Z 767.417,A -85,B 0,C 180,E1 -1621.561,E2 -1621.561} C_VEL
LIN {X 0,Y 739.331,Z 777.09,A -85,B 0,C 180,E1 -1622.036,E2 -1622.036} C_VEL
LIN {X 0,Y 739.3,Z 786.163,A -85,B 0,C 180,E1 -1622.579,E2 -1622.579} C_VEL
LIN {X 0,Y 739.249,Z 793.829,A -85,B 0,C 180,E1 -1623.123,E2 -1623.123} C_VEL
LIN {X 0,Y 739.222,Z 801.796,A -85,B 0,C 180,E1 -1623.803,E2 -1623.803} C_VEL
LIN {X 0,Y 739.182,Z 808.476,A -85,B 0,C 180,E1 -1624.484,E2 -1624.484} C_VEL
LIN {X 0,Y 739.207,Z 814.052,A -85,B 0,C 180,E1 -1625.164,E2 -1625.164} C_VEL
LIN {X 0,Y 739.181,Z 819.503,A -85,B 0,C 180,E1 -1625.983,E2 -1625.983} C_VEL
LIN {X 0,Y 739.176,Z 823.782,A -85,B 0,C 180,E1 -1626.802,E2 -1626.802} C_VEL
LIN {X 0,Y 739.168,Z 827.018,A -85,B 0,C 180,E1 -1627.623,E2 -1627.623} C_VEL
LIN {X 0,Y 739.123,Z 828.62,A -85,B 0,C 180,E1 -1628.172,E2 -1628.172} C_VEL
LIN {X 0,Y 739.172,Z 830.592,A -85,B 0,C 180,E1 -1629.27,E2 -1629.27} C_VEL
LIN {X 0,Y 739.143,Z 830.859,A -85,B 0,C 180,E1 -1630.373,E2 -1630.373} C_VEL
LIN {X 0,Y 739.13,Z 830.472,A -85,B 0,C 180,E1 -1630.925,E2 -1630.925} C_VEL
LIN {X 0,Y 739.139,Z 828.289,A -85,B 0,C 180,E1 -1632.033,E2 -1632.033} C_VEL
LIN {X 0,Y 739.153,Z 825.548,A -85,B 0,C 180,E1 -1632.867,E2 -1632.867} C_VEL
LIN {X 0,Y 739.156,Z 821.744,A -85,B 0,C 180,E1 -1633.704,E2 -1633.704} C_VEL
LIN {X 0,Y 739.19,Z 816.737,A -85,B 0,C 180,E1 -1634.543,E2 -1634.543} C_VEL
LIN {X 0,Y 739.189,Z 814.634,A -85,B 0,C 180,E1 -1634.843,E2 -1634.843} C_VEL
LIN {X 0,Y 738.569,Z 811.728,A -85,B 0,C 180,E1 -1635.239,E2 -1635.239} C_VEL
LIN {X 0,Y 735.696,Z 806.576,A -85,B 0,C 180,E1 -1635.861,E2 -1635.861} C_VEL
LIN {X 0,Y 732.823,Z 800.765,A -85,B 0,C 180,E1 -1636.449,E2 -1636.449} C_VEL
LIN {X 0,Y 732.208,Z 796.821,A -85,B 0,C 180,E1 -1636.791,E2 -1636.791} C_VEL
LIN {X 0,Y 732.252,Z 787.905,A -85,B 0,C 180,E1 -1637.465,E2 -1637.465} C_VEL
LIN {X 0,Y 732.284,Z 779.991,A -85,B 0,C 180,E1 -1637.967,E2 -1637.967} C_VEL
LIN {X 0,Y 732.328,Z 769.855,A -85,B 0,C 180,E1 -1638.498,E2 -1638.498} C_VEL
LIN {X 0,Y 732.42,Z 760.361,A -85,B 0,C 180,E1 -1638.905,E2 -1638.905} C_VEL
LIN {X 0,Y 732.417,Z 749.802,A -85,B 0,C 180,E1 -1639.265,E2 -1639.265} C_VEL
LIN {X 0,Y 732.456,Z 739.407,A -85,B 0,C 180,E1 -1639.536,E2 -1639.536} C_VEL
LIN {X 0,Y 732.537,Z 727.384,A -85,B 0,C 180,E1 -1639.752,E2 -1639.752} C_VEL
LIN {X 0,Y 732.596,Z 687.049,A -85,B 0,C 180,E1 -1640.164,E2 -1640.164} C_VEL
LIN {X 0,Y 732.466,Z 622.658,A -85,B 0,C 180,E1 -1640.794,E2 -1640.794} C_VEL
LIN {X 0,Y 732.226,Z 620.472,A -85,B 0,C 180,E1 -1640.838,E2 -1640.838} C_VEL
LIN {X 0,Y 732.325,Z 601.992,A -85,B 0,C 180,E1 -1643.475,E2 -1643.475} C_VEL
LIN {X 0,Y 732.419,Z 582.747,A -85,B 0,C 180,E1 -1646.251,E2 -1646.251} C_VEL
LIN {X 0,Y 732.443,Z 568.17,A -85,B 0,C 180,E1 -1648.38,E2 -1648.38} C_VEL
LIN {X 0,Y 732.272,Z 566.201,A -85,B 0,C 180,E1 -1648.689,E2 -1648.689} C_VEL
LIN {X 0,Y 732.285,Z 566.194,A -85,B 0,C 180,E1 -1651.099,E2 -1651.099} C_VEL
LIN {X 0,Y 732.295,Z 566.199,A -85,B 0,C 180,E1 -1653.695,E2 -1653.695} C_VEL
LIN {X 0,Y 732.256,Z 566.201,A -85,B 0,C 180,E1 -1656.374,E2 -1656.374} C_VEL
LIN {X 0,Y 732.286,Z 566.197,A -85,B 0,C 180,E1 -1658.443,E2 -1658.443} C_VEL
LIN {X 0,Y 732.31,Z 566.19,A -85,B 0,C 180,E1 -1660.92,E2 -1660.92} C_VEL
LIN {X 0,Y 732.273,Z 566.199,A -85,B 0,C 180,E1 -1663.527,E2 -1663.527} C_VEL
LIN {X 0,Y 732.299,Z 566.202,A -85,B 0,C 180,E1 -1665.838,E2 -1665.838} C_VEL
LIN {X 0,Y 732.281,Z 566.2,A -85,B 0,C 180,E1 -1668.252,E2 -1668.252} C_VEL
LIN {X 0,Y 732.3,Z 566.191,A -85,B 0,C 180,E1 -1670.854,E2 -1670.854} C_VEL
LIN {X 0,Y 732.262,Z 566.2,A -85,B 0,C 180,E1 -1673.465,E2 -1673.465} C_VEL
LIN {X 0,Y 732.289,Z 566.199,A -85,B 0,C 180,E1 -1675.643,E2 -1675.643} C_VEL
LIN {X 0,Y 732.281,Z 566.2,A -85,B 0,C 180,E1 -1677.612,E2 -1677.612} C_VEL
LIN {X 0,Y 732.285,Z 566.202,A -85,B 0,C 180,E1 -1680.172,E2 -1680.172} C_VEL
LIN {X 0,Y 732.291,Z 566.193,A -85,B 0,C 180,E1 -1682.669,E2 -1682.669} C_VEL
LIN {X 0,Y 732.294,Z 566.194,A -85,B 0,C 180,E1 -1685.323,E2 -1685.323} C_VEL
LIN {X 0,Y 732.277,Z 566.198,A -85,B 0,C 180,E1 -1687.504,E2 -1687.504} C_VEL
LIN {X 0,Y 732.297,Z 566.203,A -85,B 0,C 180,E1 -1689.858,E2 -1689.858} C_VEL
LIN {X 0,Y 732.275,Z 566.203,A -85,B 0,C 180,E1 -1692.176,E2 -1692.176} C_VEL
LIN {X 0,Y 732.28,Z 566.197,A -85,B 0,C 180,E1 -1694.465,E2 -1694.465} C_VEL
LIN {X 0,Y 732.284,Z 566.194,A -85,B 0,C 180,E1 -1696.728,E2 -1696.728} C_VEL
LIN {X 0,Y 732.299,Z 566.191,A -85,B 0,C 180,E1 -1698.971,E2 -1698.971} C_VEL
LIN {X 0,Y 732.269,Z 566.196,A -85,B 0,C 180,E1 -1701.196,E2 -1701.196} C_VEL
LIN {X 0,Y 732.298,Z 566.194,A -85,B 0,C 180,E1 -1703.409,E2 -1703.409} C_VEL
LIN {X 0,Y 732.353,Z 566.191,A -85,B 0,C 180,E1 -1705.612,E2 -1705.612} C_VEL
LIN {X 0,Y 732.338,Z 566.191,A -85,B 0,C 180,E1 -1708.356,E2 -1708.356} C_VEL
LIN {X 0,Y 732.293,Z 566.194,A -85,B 0,C 180,E1 -1710.548,E2 -1710.548} C_VEL
LIN {X 0,Y 732.27,Z 566.196,A -85,B 0,C 180,E1 -1712.741,E2 -1712.741} C_VEL
LIN {X 0,Y 732.347,Z 566.185,A -85,B 0,C 180,E1 -1714.938,E2 -1714.938} C_VEL
LIN {X 0,Y 732.321,Z 566.189,A -85,B 0,C 180,E1 -1717.143,E2 -1717.143} C_VEL
LIN {X 0,Y 732.313,Z 566.202,A -85,B 0,C 180,E1 -1719.914,E2 -1719.914} C_VEL
LIN {X 0,Y 732.314,Z 566.19,A -85,B 0,C 180,E1 -1722.708,E2 -1722.708} C_VEL
LIN {X 0,Y 732.325,Z 566.188,A -85,B 0,C 180,E1 -1724.979,E2 -1724.979} C_VEL
LIN {X 0,Y 732.303,Z 566.192,A -85,B 0,C 180,E1 -1727.248,E2 -1727.248} C_VEL
LIN {X 0,Y 732.282,Z 566.199,A -85,B 0,C 180,E1 -1729.559,E2 -1729.559} C_VEL
LIN {X 0,Y 732.3,Z 566.204,A -85,B 0,C 180,E1 -1731.906,E2 -1731.906} C_VEL
LIN {X 0,Y 732.263,Z 566.202,A -85,B 0,C 180,E1 -1734.287,E2 -1734.287} C_VEL
LIN {X 0,Y 732.284,Z 566.194,A -85,B 0,C 180,E1 -1736.716,E2 -1736.716} C_VEL
LIN {X 0,Y 732.293,Z 566.193,A -85,B 0,C 180,E1 -1739.197,E2 -1739.197} C_VEL
LIN {X 0,Y 732.29,Z 566.199,A -85,B 0,C 180,E1 -1741.648,E2 -1741.648} C_VEL
LIN {X 0,Y 732.292,Z 566.2,A -85,B 0,C 180,E1 -1743.695,E2 -1743.695} C_VEL
LIN {X 0,Y 732.264,Z 566.2,A -85,B 0,C 180,E1 -1746.374,E2 -1746.374} C_VEL
LIN {X 0,Y 732.287,Z 566.196,A -85,B 0,C 180,E1 -1748.443,E2 -1748.443} C_VEL
LIN {X 0,Y 732.313,Z 566.19,A -85,B 0,C 180,E1 -1750.921,E2 -1750.921} C_VEL
LIN {X 0,Y 732.271,Z 566.2,A -85,B 0,C 180,E1 -1753.528,E2 -1753.528} C_VEL
LIN {X 0,Y 732.296,Z 566.203,A -85,B 0,C 180,E1 -1755.838,E2 -1755.838} C_VEL
LIN {X 0,Y 732.279,Z 566.201,A -85,B 0,C 180,E1 -1758.253,E2 -1758.253} C_VEL
LIN {X 0,Y 732.308,Z 566.19,A -85,B 0,C 180,E1 -1760.856,E2 -1760.856} C_VEL
LIN {X 0,Y 732.256,Z 566.201,A -85,B 0,C 180,E1 -1763.466,E2 -1763.466} C_VEL
LIN {X 0,Y 732.285,Z 566.2,A -85,B 0,C 180,E1 -1765.644,E2 -1765.644} C_VEL
LIN {X 0,Y 732.284,Z 566.2,A -85,B 0,C 180,E1 -1768.259,E2 -1768.259} C_VEL
LIN {X 0,Y 732.276,Z 566.195,A -85,B 0,C 180,E1 -1770.802,E2 -1770.802} C_VEL
LIN {X 0,Y 732.254,Z 566.199,A -85,B 0,C 180,E1 -1773.283,E2 -1773.283} C_VEL
LIN {X 0,Y 732.258,Z 566.205,A -85,B 0,C 180,E1 -1775.713,E2 -1775.713} C_VEL
LIN {X 0,Y 732.289,Z 566.203,A -85,B 0,C 180,E1 -1778.097,E2 -1778.097} C_VEL
LIN {X 0,Y 732.278,Z 566.197,A -85,B 0,C 180,E1 -1780.441,E2 -1780.441} C_VEL
LIN {X 0,Y 732.296,Z 566.192,A -85,B 0,C 180,E1 -1783.039,E2 -1783.039} C_VEL
LIN {X 0,Y 732.275,Z 566.2,A -85,B 0,C 180,E1 -1785.6,E2 -1785.6} C_VEL
LIN {X 0,Y 732.297,Z 566.203,A -85,B 0,C 180,E1 -1787.853,E2 -1787.853} C_VEL
LIN {X 0,Y 732.321,Z 566.19,A -85,B 0,C 180,E1 -1790.642,E2 -1790.642} C_VEL
LIN {X 0,Y 732.288,Z 566.193,A -85,B 0,C 180,E1 -1792.857,E2 -1792.857} C_VEL
LIN {X 0,Y 732.312,Z 566.19,A -85,B 0,C 180,E1 -1795.062,E2 -1795.062} C_VEL
LIN {X 0,Y 732.329,Z 566.198,A -85,B 0,C 180,E1 -1797.808,E2 -1797.808} C_VEL
LIN {X 0,Y 732.302,Z 566.193,A -85,B 0,C 180,E1 -1800.548,E2 -1800.548} C_VEL
LIN {X 0,Y 732.265,Z 566.196,A -85,B 0,C 180,E1 -1802.742,E2 -1802.742} C_VEL
LIN {X 0,Y 732.324,Z 566.188,A -85,B 0,C 180,E1 -1804.938,E2 -1804.938} C_VEL
LIN {X 0,Y 732.278,Z 566.195,A -85,B 0,C 180,E1 -1807.143,E2 -1807.143} C_VEL
LIN {X 0,Y 732.308,Z 566.193,A -85,B 0,C 180,E1 -1809.358,E2 -1809.358} C_VEL
LIN {X 0,Y 732.254,Z 566.203,A -85,B 0,C 180,E1 -1811.588,E2 -1811.588} C_VEL
LIN {X 0,Y 732.275,Z 566.196,A -85,B 0,C 180,E1 -1813.272,E2 -1813.272} C_VEL
LIN {X 0,Y 732.273,Z 566.2,A -85,B 0,C 180,E1 -1815.535,E2 -1815.535} C_VEL
LIN {X 0,Y 732.264,Z 566.207,A -85,B 0,C 180,E1 -1817.824,E2 -1817.824} C_VEL
LIN {X 0,Y 732.285,Z 566.197,A -85,B 0,C 180,E1 -1820.383,E2 -1820.383} C_VEL
LIN {X 0,Y 732.256,Z 566.199,A -85,B 0,C 180,E1 -1822.496,E2 -1822.496} C_VEL
LIN {X 0,Y 732.27,Z 566.195,A -85,B 0,C 180,E1 -1824.89,E2 -1824.89} C_VEL
LIN {X 0,Y 732.28,Z 566.196,A -85,B 0,C 180,E1 -1827.331,E2 -1827.331} C_VEL
LIN {X 0,Y 732.276,Z 566.205,A -85,B 0,C 180,E1 -1829.828,E2 -1829.828} C_VEL
LIN {X 0,Y 732.251,Z 566.201,A -85,B 0,C 180,E1 -1832.39,E2 -1832.39} C_VEL
LIN {X 0,Y 732.263,Z 566.197,A -85,B 0,C 180,E1 -1834.651,E2 -1834.651} C_VEL
LIN {X 0,Y 732.257,Z 566.2,A -85,B 0,C 180,E1 -1837.445,E2 -1837.445} C_VEL
LIN {X 0,Y 732.24,Z 566.211,A -85,B 0,C 180,E1 -1839.859,E2 -1839.859} C_VEL
LIN {X 0,Y 732.257,Z 566.208,A -85,B 0,C 180,E1 -1842.035,E2 -1842.035} C_VEL
LIN {X 0,Y 732.285,Z 566.199,A -85,B 0,C 180,E1 -1844.287,E2 -1844.287} C_VEL
LIN {X 0,Y 732.246,Z 566.199,A -85,B 0,C 180,E1 -1846.635,E2 -1846.635} C_VEL
LIN {X 0,Y 732.27,Z 566.195,A -85,B 0,C 180,E1 -1849.083,E2 -1849.083} C_VEL
LIN {X 0,Y 732.274,Z 566.202,A -85,B 0,C 180,E1 -1851.661,E2 -1851.661} C_VEL
LIN {X 0,Y 732.243,Z 566.202,A -85,B 0,C 180,E1 -1854.398,E2 -1854.398} C_VEL
LIN {X 0,Y 732.263,Z 566.196,A -85,B 0,C 180,E1 -1856.96,E2 -1856.96} C_VEL
LIN {X 0,Y 732.252,Z 566.202,A -85,B 0,C 180,E1 -1859.537,E2 -1859.537} C_VEL
LIN {X 0,Y 732.254,Z 566.208,A -85,B 0,C 180,E1 -1862.049,E2 -1862.049} C_VEL
LIN {X 0,Y 732.252,Z 566.201,A -85,B 0,C 180,E1 -1864.504,E2 -1864.504} C_VEL
LIN {X 0,Y 732.227,Z 566.202,A -85,B 0,C 180,E1 -1866.908,E2 -1866.908} C_VEL
LIN {X 0,Y 732.272,Z 566.338,A -85,B 0,C 180,E1 -1868.961,E2 -1868.961} C_VEL
LIN {X 0,Y 732.676,Z 571.469,A -85,B 0,C 180,E1 -1869.623,E2 -1869.623} C_VEL
LIN {X 0,Y 732.569,Z 590.776,A -85,B 0,C 180,E1 -1872.04,E2 -1872.04} C_VEL
LIN {X 0,Y 732.398,Z 611.715,A -85,B 0,C 180,E1 -1874.624,E2 -1874.624} C_VEL
LIN {X 0,Y 732.312,Z 630.108,A -85,B 0,C 180,E1 -1876.87,E2 -1876.87} C_VEL
LIN {X 0,Y 732.234,Z 647.461,A -85,B 0,C 180,E1 -1878.97,E2 -1878.97} C_VEL
LIN {X 0,Y 732.22,Z 649.485,A -85,B 0,C 180,E1 -1879.214,E2 -1879.214} C_VEL
LIN {X 0,Y 732.62,Z 656.457,A -85,B 0,C 180,E1 -1879.29,E2 -1879.29} C_VEL
LIN {X 0,Y 732.481,Z 755.852,A -85,B 0,C 180,E1 -1880.275,E2 -1880.275} C_VEL
LIN {X 0,Y 732.468,Z 765.421,A -85,B 0,C 180,E1 -1880.429,E2 -1880.429} C_VEL
LIN {X 0,Y 732.431,Z 776.186,A -85,B 0,C 180,E1 -1880.678,E2 -1880.678} C_VEL
LIN {X 0,Y 732.444,Z 786.28,A -85,B 0,C 180,E1 -1880.991,E2 -1880.991} C_VEL
LIN {X 0,Y 732.376,Z 796.775,A -85,B 0,C 180,E1 -1881.406,E2 -1881.406} C_VEL
LIN {X 0,Y 732.307,Z 806.622,A -85,B 0,C 180,E1 -1881.89,E2 -1881.89} C_VEL
LIN {X 0,Y 732.237,Z 815.846,A -85,B 0,C 180,E1 -1882.442,E2 -1882.442} C_VEL
LIN {X 0,Y 732.226,Z 823.584,A -85,B 0,C 180,E1 -1882.995,E2 -1882.995} C_VEL
LIN {X 0,Y 732.164,Z 831.633,A -85,B 0,C 180,E1 -1883.684,E2 -1883.684} C_VEL
LIN {X 0,Y 732.108,Z 838.197,A -85,B 0,C 180,E1 -1884.355,E2 -1884.355} C_VEL
LIN {X 0,Y 732.147,Z 843.953,A -85,B 0,C 180,E1 -1885.061,E2 -1885.061} C_VEL
LIN {X 0,Y 732.127,Z 849.403,A -85,B 0,C 180,E1 -1885.885,E2 -1885.885} C_VEL
LIN {X 0,Y 732.074,Z 853.688,A -85,B 0,C 180,E1 -1886.709,E2 -1886.709} C_VEL
LIN {X 0,Y 732.092,Z 855.974,A -85,B 0,C 180,E1 -1887.258,E2 -1887.258} C_VEL
LIN {X 0,Y 732.031,Z 859.199,A -85,B 0,C 180,E1 -1888.355,E2 -1888.355} C_VEL
LIN {X 0,Y 732.039,Z 860.715,A -85,B 0,C 180,E1 -1889.452,E2 -1889.452} C_VEL
LIN {X 0,Y 732.038,Z 861,A -85,B 0,C 180,E1 -1890,E2 -1890} C_VEL
LIN {X 0,Y 732.041,Z 860.143,A -85,B 0,C 180,E1 -1891.097,E2 -1891.097} C_VEL
LIN {X 0,Y 732.032,Z 859.199,A -85,B 0,C 180,E1 -1891.645,E2 -1891.645} C_VEL
LIN {X 0,Y 732.092,Z 855.974,A -85,B 0,C 180,E1 -1892.742,E2 -1892.742} C_VEL
LIN {X 0,Y 732.081,Z 852.423,A -85,B 0,C 180,E1 -1893.566,E2 -1893.566} C_VEL
LIN {X 0,Y 732.064,Z 847.765,A -85,B 0,C 180,E1 -1894.39,E2 -1894.39} C_VEL
LIN {X 0,Y 732.161,Z 841.853,A -85,B 0,C 180,E1 -1895.215,E2 -1895.215} C_VEL
LIN {X 0,Y 732.176,Z 834.463,A -85,B 0,C 180,E1 -1896.041,E2 -1896.041} C_VEL
LIN {X 0,Y 732.213,Z 826.97,A -85,B 0,C 180,E1 -1896.73,E2 -1896.73} C_VEL
LIN {X 0,Y 732.264,Z 818.879,A -85,B 0,C 180,E1 -1897.351,E2 -1897.351} C_VEL
LIN {X 0,Y 732.302,Z 810.27,A -85,B 0,C 180,E1 -1897.903,E2 -1897.903} C_VEL
LIN {X 0,Y 732.349,Z 801.228,A -85,B 0,C 180,E1 -1898.387,E2 -1898.387} C_VEL
LIN {X 0,Y 732.395,Z 791.833,A -85,B 0,C 180,E1 -1898.802,E2 -1898.802} C_VEL
LIN {X 0,Y 732.418,Z 780.978,A -85,B 0,C 180,E1 -1899.183,E2 -1899.183} C_VEL
LIN {X 0,Y 732.465,Z 769.81,A -85,B 0,C 180,E1 -1899.479,E2 -1899.479} C_VEL
LIN {X 0,Y 732.495,Z 759.273,A -85,B 0,C 180,E1 -1899.679,E2 -1899.679} C_VEL
LIN {X 0,Y 732.512,Z 741.647,A -85,B 0,C 180,E1 -1899.88,E2 -1899.88} C_VEL
LIN {X 0,Y 732.489,Z 651.534,A -85,B 0,C 180,E1 -1900.76,E2 -1900.76} C_VEL
LIN {X 0,Y 732.22,Z 649.483,A -85,B 0,C 180,E1 -1900.786,E2 -1900.786} C_VEL
LIN {X 0,Y 732.309,Z 631.263,A -85,B 0,C 180,E1 -1902.99,E2 -1902.99} C_VEL
LIN {X 0,Y 732.403,Z 612.985,A -85,B 0,C 180,E1 -1905.22,E2 -1905.22} C_VEL
LIN {X 0,Y 732.54,Z 593.088,A -85,B 0,C 180,E1 -1907.673,E2 -1907.673} C_VEL
LIN {X 0,Y 732.669,Z 573.422,A -85,B 0,C 180,E1 -1910.131,E2 -1910.131} C_VEL
LIN {X 0,Y 732.53,Z 567.638,A -85,B 0,C 180,E1 -1910.866,E2 -1910.866} C_VEL
LIN {X 0,Y 732.262,Z 566.205,A -85,B 0,C 180,E1 -1911.058,E2 -1911.058} C_VEL
LIN {X 0,Y 732.219,Z 566.211,A -85,B 0,C 180,E1 -1913.689,E2 -1913.689} C_VEL
LIN {X 0,Y 732.261,Z 566.206,A -85,B 0,C 180,E1 -1916.105,E2 -1916.105} C_VEL
LIN {X 0,Y 732.241,Z 566.201,A -85,B 0,C 180,E1 -1918.574,E2 -1918.574} C_VEL
LIN {X 0,Y 732.264,Z 566.198,A -85,B 0,C 180,E1 -1920.583,E2 -1920.583} C_VEL
LIN {X 0,Y 732.282,Z 566.197,A -85,B 0,C 180,E1 -1923.04,E2 -1923.04} C_VEL
LIN {X 0,Y 732.284,Z 566.204,A -85,B 0,C 180,E1 -1925.696,E2 -1925.696} C_VEL
LIN {X 0,Y 732.283,Z 566.194,A -85,B 0,C 180,E1 -1928.443,E2 -1928.443} C_VEL
LIN {X 0,Y 732.3,Z 566.202,A -85,B 0,C 180,E1 -1931.299,E2 -1931.299} C_VEL
LIN {X 0,Y 732.296,Z 566.193,A -85,B 0,C 180,E1 -1934.287,E2 -1934.287} C_VEL
LIN {X 0,Y 732.275,Z 566.198,A -85,B 0,C 180,E1 -1936.633,E2 -1936.633} C_VEL
LIN {X 0,Y 732.317,Z 566.201,A -85,B 0,C 180,E1 -1939.08,E2 -1939.08} C_VEL
LIN {X 0,Y 732.292,Z 566.196,A -85,B 0,C 180,E1 -1941.66,E2 -1941.66} C_VEL
LIN {X 0,Y 732.296,Z 566.195,A -85,B 0,C 180,E1 -1944.393,E2 -1944.393} C_VEL
LIN {X 0,Y 732.304,Z 566.204,A -85,B 0,C 180,E1 -1946.962,E2 -1946.962} C_VEL
LIN {X 0,Y 732.278,Z 566.196,A -85,B 0,C 180,E1 -1949.538,E2 -1949.538} C_VEL
LIN {X 0,Y 732.284,Z 566.195,A -85,B 0,C 180,E1 -1952.05,E2 -1952.05} C_VEL
LIN {X 0,Y 732.288,Z 566.203,A -85,B 0,C 180,E1 -1954.505,E2 -1954.505} C_VEL
LIN {X 0,Y 732.267,Z 566.203,A -85,B 0,C 180,E1 -1956.91,E2 -1956.91} C_VEL
LIN {X 0,Y 732.288,Z 566.195,A -85,B 0,C 180,E1 -1959.273,E2 -1959.273} C_VEL
LIN {X 0,Y 732.302,Z 566.193,A -85,B 0,C 180,E1 -1961.6,E2 -1961.6} C_VEL
LIN {X 0,Y 732.303,Z 566.196,A -85,B 0,C 180,E1 -1963.896,E2 -1963.896} C_VEL
LIN {X 0,Y 732.271,Z 566.206,A -85,B 0,C 180,E1 -1966.164,E2 -1966.164} C_VEL
LIN {X 0,Y 732.263,Z 566.207,A -85,B 0,C 180,E1 -1968.412,E2 -1968.412} C_VEL
LIN {X 0,Y 732.311,Z 566.198,A -85,B 0,C 180,E1 -1970.642,E2 -1970.642} C_VEL
LIN {X 0,Y 732.311,Z 566.357,A -85,B 0,C 180,E1 -1971.439,E2 -1971.439} C_VEL
LIN {X 0,Y 732.403,Z 579.799,A -85,B 0,C 180,E1 -1973.41,E2 -1973.41} C_VEL
LIN {X 0,Y 732.329,Z 596.917,A -85,B 0,C 180,E1 -1975.886,E2 -1975.886} C_VEL
LIN {X 0,Y 732.227,Z 614.172,A -85,B 0,C 180,E1 -1978.355,E2 -1978.355} C_VEL
LIN {X 0,Y 732.234,Z 620.552,A -85,B 0,C 180,E1 -1979.263,E2 -1979.263} C_VEL
LIN {X 0,Y 732.649,Z 626.12,A -85,B 0,C 180,E1 -1979.332,E2 -1979.332} C_VEL
LIN {X 0,Y 732.457,Z 726.498,A -85,B 0,C 180,E1 -1980.325,E2 -1980.325} C_VEL
LIN {X 0,Y 732.421,Z 738.314,A -85,B 0,C 180,E1 -1980.531,E2 -1980.531} C_VEL
LIN {X 0,Y 732.405,Z 748.502,A -85,B 0,C 180,E1 -1980.788,E2 -1980.788} C_VEL
LIN {X 0,Y 732.424,Z 757.976,A -85,B 0,C 180,E1 -1981.096,E2 -1981.096} C_VEL
LIN {X 0,Y 732.346,Z 768.042,A -85,B 0,C 180,E1 -1981.507,E2 -1981.507} C_VEL
LIN {X 0,Y 732.294,Z 777.604,A -85,B 0,C 180,E1 -1981.987,E2 -1981.987} C_VEL
LIN {X 0,Y 732.254,Z 786.589,A -85,B 0,C 180,E1 -1982.535,E2 -1982.535} C_VEL
LIN {X 0,Y 732.178,Z 795.034,A -85,B 0,C 180,E1 -1983.153,E2 -1983.153} C_VEL
LIN {X 0,Y 732.156,Z 802.802,A -85,B 0,C 180,E1 -1983.84,E2 -1983.84} C_VEL
LIN {X 0,Y 732.094,Z 809.317,A -85,B 0,C 180,E1 -1984.527,E2 -1984.527} C_VEL
LIN {X 0,Y 732.119,Z 814.738,A -85,B 0,C 180,E1 -1985.215,E2 -1985.215} C_VEL
LIN {X 0,Y 732.106,Z 820.047,A -85,B 0,C 180,E1 -1986.041,E2 -1986.041} C_VEL
LIN {X 0,Y 732.082,Z 824.196,A -85,B 0,C 180,E1 -1986.869,E2 -1986.869} C_VEL
LIN {X 0,Y 732.072,Z 827.31,A -85,B 0,C 180,E1 -1987.698,E2 -1987.698} C_VEL
LIN {X 0,Y 732.036,Z 828.883,A -85,B 0,C 180,E1 -1988.252,E2 -1988.252} C_VEL
LIN {X 0,Y 732.075,Z 830.666,A -85,B 0,C 180,E1 -1989.361,E2 -1989.361} C_VEL
LIN {X 0,Y 732.067,Z 830.962,A -85,B 0,C 180,E1 -1989.917,E2 -1989.917} C_VEL
LIN {X 0,Y 732.055,Z 830.35,A -85,B 0,C 180,E1 -1991.032,E2 -1991.032} C_VEL
LIN {X 0,Y 732.059,Z 829.396,A -85,B 0,C 180,E1 -1991.591,E2 -1991.591} C_VEL
LIN {X 0,Y 732.069,Z 826.273,A -85,B 0,C 180,E1 -1992.713,E2 -1992.713} C_VEL
LIN {X 0,Y 732.074,Z 822.706,A -85,B 0,C 180,E1 -1993.557,E2 -1993.557} C_VEL
LIN {X 0,Y 732.095,Z 817.983,A -85,B 0,C 180,E1 -1994.404,E2 -1994.404} C_VEL
LIN {X 0,Y 732.13,Z 811.923,A -85,B 0,C 180,E1 -1995.254,E2 -1995.254} C_VEL
LIN {X 0,Y 732.12,Z 804.269,A -85,B 0,C 180,E1 -1996.108,E2 -1996.108} C_VEL
LIN {X 0,Y 732.208,Z 796.821,A -85,B 0,C 180,E1 -1996.791,E2 -1996.791} C_VEL
LIN {X 0,Y 731.607,Z 792.812,A -85,B 0,C 180,E1 -1997.121,E2 -1997.121} C_VEL
LIN {X 0,Y 728.799,Z 785.887,A -85,B 0,C 180,E1 -1997.639,E2 -1997.639} C_VEL
LIN {X 0,Y 725.955,Z 778.588,A -85,B 0,C 180,E1 -1998.12,E2 -1998.12} C_VEL
LIN {X 0,Y 725.307,Z 773.799,A -85,B 0,C 180,E1 -1998.39,E2 -1998.39} C_VEL
